(* Schneider Machine Expert - Basic project Bex CT 03 August 2023, file version 2.8.0.0 *)
(* ProjectInformations: Name=New project *)

HARDWARE
  Cpu 0: TM221CE40R
  EthernetConfiguration: NetworkName=M221, IpAllocationMode=FixedAddress, IpAddress=192.168.1.10, SubnetMask=255.255.255.0
  SerialLineConfiguration: Baud=Baud19200, Parity=ParityEven, DataBits=DataBits8, StopBits=StopBits1, PhysicalMedium=PhysicalMediumRs232, TransmissionMode=TransmissionModeModbusRtu, SlaveId=1, Addressing=MasterAddressing
  MastTask: UsePeriodScanMode=false, PeriodScan=100
  FastTask: Period=255
  CpuBehavior: StartingMode=StartAsPreviousState, AutoSaveRamOnEeprom=true, WatchdogPeriod=250

SYMBOLS  (address, symbol, comment, settings)
  %M0       SU_ALARM_AUX  "START UP ALARM AUX BIT"
  %M1       TRIP_ALARM_AUX  "SAFTY ALARM AUX BIT"
  %M2       C1_TRIP  "CONVEYOR No1 VSD TRIP"
  %M3       C2_TRIP  "CONVEYOR No2 VSD TRIP"
  %M4       SC1_TRIP  "SCALE CONVEYOR No1 VSD TRIP"
  %M5       SC1_FAULT_CONT  "SCALE CONTROL FAULT"
  %M6       C3_TRIP  "CONVEYOR No3 VSD TRIP"
  %M7       NO_PROD_STOP  "NO PRODUCT ON CONVEYOR 1 FOR PRE SET TIME"
  %M8       STOP_AUX_BIT  "STOP SEQUENCE ENERGISED"
  %M9       E_STOP_BIT  "EMERGENCY STOP AUX BIT"
  %M10      HEALTHY_BIT  "SYSTEM HEALTHY"
  %M11      C1_AUTO_START  "CONVEYOR 1 AUTO START BIT"
  %M12      C2_AUTO_START  "CONVEYOR 2 AUTO START BIT"
  %M13      SC1_AUTO_START  "SCALE CONVEYOR 1 AUTO START BIT"
  %M14      C3_AUTO_START  "CONVEYOR 3 AUTO START BIT"
  %M15      SYY_AUTO_ON  "SYSTEM AUTO RUNNING"
  %M16      C2_AUTO_STOP  "CONVEYOR 2 AUTO STOP BIT"
  %M17      SC1_AUTO_STOP  "SCALE CONVEYOR 1 AUTO STOP BIT"
  %M18      C3_AUTO_STOP  "CONVEYOR 3 AUTO STOP BIT"
  %M19      AUTO_ON_STOP  "AUTO STOP SEQUENCE ON"
  %M20      C1_ON_AUX  "C1 CONTROL BIT FULL SPEED"
  %M21      C1_ON_SLOW_AUX  "C1 CONTROL BIT SLOW SPEED"
  %M22      C2_ON_AUX  "C2 CONTROL BIT FULL SPEED"
  %M23      SC1_ON_AUX  "SC1 CONTROL BIT FULL SPEED"
  %M24      C3_ON_AUX  "C3 CONTROL BIT FULL SPEED"
  %M25      BAD_READ_AUX  "PRODUCT NOT SCANED"
  %M26      C1A_FAULT  "C1 PHOTO CELL NOT WORKING"
  %M27      C2A_FAULT  "C2 PHOTO CELL NOT WORKING"
  %M28      SC1A_FAULT  "SC1 PHOTO CELL NOT WORKING"
  %M29      C3A_FAULT  "C3 PHOTO CELL NOT WORKING"
  %M30      C1_PROD_TO_CLOSE  "PRODUCT TO CLOSED ON C1"
  %M31      C1_RESTART_PTC  "RESTART C1 AFTER PRODUCT HAS RECH CORECT DISTANCE"
  %M32      C2_PROD_TO_CLOSED  "PRODUCT TO CLOSED ON C2"
  %M33      C2_RESTART_PTC  "RESTART C2 AFTER PRODUCT HAS RECH CORECT DISTANCE"
  %M34      C1_RESTART_DELAY_C2  "RESTART C1 AFTER C2 START - TIME DELAY BIT"
  %M35      C1_RESTART_C2  "RESTART C1 AFTER C2 START - COMMAND BIT"
  %M36      SYS_RESTART_AFTER_BAD_READ  "SYSTEM RESTARTING AFTER BAD READ - AUX BIT"
  %M37      RESET_COUNTER_2  "RESET BIT FOR PRODUCT DISTANCE ON C2"
  %M38      C1A_SET_BIT  "PRODUCT COUNTER ON C1 (DISTANCE OF THE PRODUCT)"
  %M39      C2A_SET_BIT  "PRODUCT COUNTER ON C2 (DISTANCE OF THE PRODUCT)"
  %M40      APP_ON  "SIGNAL SEND FROM PC - APP ON"
  %M41      GOOD_READ_HSCAN  "SIGNAL SEND FROM THE PC - HAND SCAN GOOD READ AUX BIT"
  %M42      STOP_RUN_MSG
  %M43      HS_RESTART  "SCANING THE PRODUCT WITH HAND SCAN - GOOD READ"
  %M44      C3_BAD_READ_DELAY
  %M45      SC1A_ACTIVE_AUX1
  %M46      SCALE_EMPTY
  %M47      C1_RESTART_TIME_OUT
  %M48      C1_C2_STOP_INTERLOCK
  %M49      CF_STO_BIT
  %M50      RUN_IND
  %M51      STOP_IND
  %M52      SCALE_EMPTY_AUX
  %M53      SCALE_EMPTY_AUX1
  %M54      APP_ON_SUP_DELAY
  %M55      C2A_ACTIVE_AUX
  %M56      C2A_ACTIVE_RESET
  %M57      BAD_READ_AL
  %M58      BAD_READ_AL_AUX
  %M59      APP_SUP_DELAY_STOP
  %M60      C2_STOP_BAD_READ
  %M61      C1_STOP_BAD_READ
  %M255     BA_PASS_BIT
  %S6       SB_TB1S  "Time base of 1 s generated by an internal clock"
  %S112     SB_IOSCANETHRESET  "Set to 1 to reset the IOScanner on Ethernet"
  %SW212    SW_IOSCANETHSTATUS  "Contains the IOScanner status on Ethernet"
  %MW10     FAULT_ALARM_01  "TRIP/ALARM  SIGNALS SEND TO PC"
  %MW11     RUN_STOP_TO_PC  "SYSTEM RUNNING / STOP   SIGNALS SEND TO PC"
  %MW12     SC1A_TO_PC  "SCALE PHOTO SENSOR SC1A SIGNAL SEND TO PC"
  %MW14     PC_ON_RECEIVED
  %MW20     RECEIVED_FROM_PC_ON  "SIGNAL SEND FROM PC - PC ON"
  %MW25     RECEIVED_FROM_PC_HSGR  "SIGNAL RECEIVED FROM PC - HAND SCAN GOOD READ"
  %TM0        [Preset=14, Base=OneSecond]
  %TM1        [Preset=10]
  %TM2        [Preset=25, Base=OneSecond]
  %TM3        [Preset=100, Base=OneSecond]
  %TM4        [Preset=1, Base=OneSecond]
  %TM5        [Preset=1, Base=OneSecond]
  %TM6        [Preset=5, Base=TenMilliSeconds]
  %TM7        [Preset=2, Base=TenMilliSeconds]
  %TM8        [Preset=180, Base=OneSecond]
  %TM9        [Preset=180, Base=OneSecond]
  %TM10       [Preset=180, Base=OneSecond]
  %TM11       [Preset=120, Base=OneSecond]
  %TM12       [Preset=1, Base=OneSecond]
  %TM13       [Preset=30, Base=TenMilliSeconds]
  %TM14       [Preset=3, Base=OneSecond]
  %TM15       [Type=TOF, Preset=120, Base=OneSecond]
  %TM16       [Preset=1, Base=TenMilliSeconds]
  %TM17       [Preset=3, Base=OneSecond]
  %TM18       [Preset=3, Base=OneSecond]
  %TM19       [Preset=5, Base=TenMilliSeconds]
  %TM20       [Preset=5, Base=TenMilliSeconds]
  %C0         [Preset=2]
  %C1         [Preset=2]
  %I0.0     E_STOP_PB  "EMERGENCY STOP PUSH BUTTON"
  %I0.1     SYS_START_PB  "Alarm Acknowledge Push Button"
  %I0.2     SYS_STOP_PB  "Alarm Reset Push Button"
  %I0.3     ALARM_ACKG  "System Start Push Button"
  %I0.4     ALARM_RESET  "System Stop Push Button"
  %I0.5     C1_RUNNING  "Conveyor No.1 Running  VSD"
  %I0.6     C2_RUNNING  "Conveyor No.2 Running  VSD"
  %I0.7     SC1_RUNNING  "Scale Conveyor No.1 Running  VSD"
  %I0.8     C3_RUNNING  "Conveyor No.3 Running  VSD"
  %I0.9     C1A_ACTIVE  "Conveyor No.1 Photo Sensor"
  %I0.10    C2A_ACTIVE  "Conveyor No.2 Photo Sensor"
  %I0.11    SC1A_ACTIVE  "Scale Conveyor No.1 Photo Sensor"
  %I0.12    SC1B_ACTIVE  "Scale Conveyor No.1  Control Fault"
  %I0.13    C3A_ACTIVE  "Conveyor No.3 Photo Sensor"
  %I0.14    GOOD_READ_ACTIVE  "Camera Product Good Read"
  %I0.15    BAD_READ_ACTIVE  "Camera Product Bad Read"
  %I0.16    LASER_READ  "LASER SIGNAL IN"
  %I0.17    CAMERA_SENS  "CAMERA SENSOR ON SCALE CONVEYOR"
  %Q0.0     C1_ON  "Conveyor No.1 - ON/OFF Fast"
  %Q0.1     C1_ON_SLOW  "Conveyor No.1 - SLOW SPEED"
  %Q0.2     C2_ON  "Conveyor No.2 - ON/OFF Fast"
  %Q0.3     C2_ON_SLOW  "Conveyor No.2 - SLOW SPEED"
  %Q0.4     SC1_ON  "Scale belt No.1 - ON/OFF Fast"
  %Q0.5     SC1_ON_SLOW  "Scale belt No.1 - SLOW SPEED"
  %Q0.6     C3_ON  "ConveConveyor No.3 - ON/OFF Fast"
  %Q0.7     C3_ON_SLOW  "Conveyor No.3 - SLOW SPEED"
  %Q0.8     SYS_RUNNING_IND  "System Running Green Indication"
  %Q0.9     SYS_TRIP_IND  "System Trip Red Indication"
  %Q0.10    ALARM_BUZZER  "Alarm Buzzer"
  %Q0.11    GOOD_READ_IND  "Product Good read Tower Green indication"
  %Q0.12    BAD_READ_IND  "Product Bad read Tower Green indication"
  %Q0.13    SC1_CONT_ON  "Start Scale - Signal to Scale Control  Panel"
  %Q0.14    CAM_TRIGGER  "Camera On/Off with laser or Sensor on the scale belt"
  %Q0.15    COLLING_FAN
  %IWN300.0.0 PC_IN_01  "APPLICATION RUNNING / STOP SIGNAL SEND FROM THE PC"  [Channel=Device 1_Channel0]
  %IWN300.0.1 PC_IN_02  "HAND SCANER ON/OFF SIGNAL SEND FROM PC"  [Channel=Device 1_Channel0]
  %QWN300.1.0 PC_OUT_01  "SENDING TO PC - ALARMS"  [Channel=Device 1_Channel1]
  %QWN300.1.1 PC_OUT_02  "SENDING TO PC STATUS (RUN, STOP, E/STOP)"  [Channel=Device 1_Channel1]
  %QWN300.1.2 PC_OUT_03  "SENDING TO PC - SCALE PHOTO SENSOR STATUS"  [Channel=Device 1_Channel1]
  %QWN300.1.3 PC_OUT_04  [Channel=Device 1_Channel1]

POU GENERAL ALARM
  (* SectionNumber=1 *)

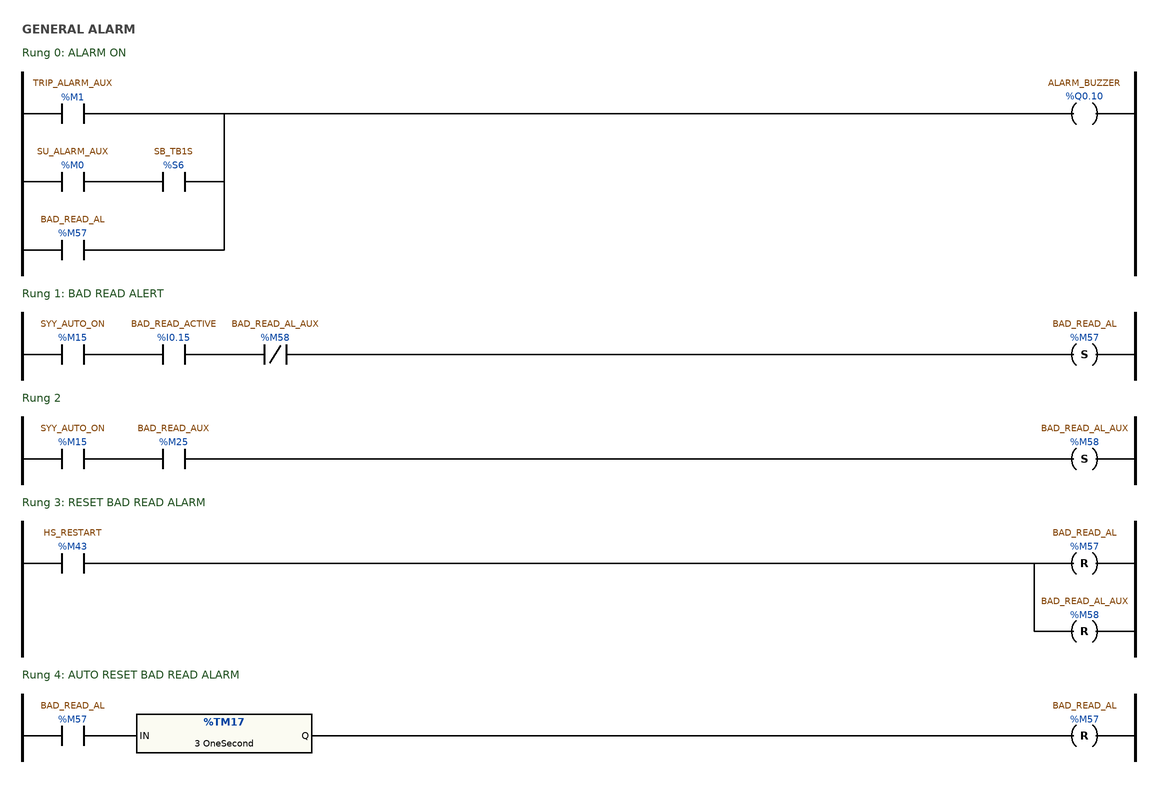

// Rung 0: ALARM ON
  LD %M1                  (* TRIP_ALARM_AUX *)
  OR( %M0                 (* SU_ALARM_AUX *)
  AND %S6                 (* SB_TB1S *)
  )
  OR %M57                 (* BAD_READ_AL *)
  ST %Q0.10               (* ALARM_BUZZER *)
  // as ST:
  //   ALARM_BUZZER := TRIP_ALARM_AUX OR SU_ALARM_AUX AND SB_TB1S OR BAD_READ_AL;

// Rung 1: BAD READ ALERT
  LD %M15                 (* SYY_AUTO_ON *)
  AND %I0.15              (* BAD_READ_ACTIVE *)
  ANDN %M58               (* BAD_READ_AL_AUX *)
  S %M57                  (* BAD_READ_AL *)
  // as ST:
  //   IF SYY_AUTO_ON AND BAD_READ_ACTIVE AND NOT BAD_READ_AL_AUX THEN BAD_READ_AL := TRUE; END_IF;

// Rung 2
  LD %M15                 (* SYY_AUTO_ON *)
  AND %M25                (* BAD_READ_AUX *)
  S %M58                  (* BAD_READ_AL_AUX *)
  // as ST:
  //   IF SYY_AUTO_ON AND BAD_READ_AUX THEN BAD_READ_AL_AUX := TRUE; END_IF;

// Rung 3: RESET BAD READ ALARM
  LD %M43                 (* HS_RESTART *)
  R %M57                  (* BAD_READ_AL *)
  R %M58                  (* BAD_READ_AL_AUX *)
  // as ST:
  //   IF HS_RESTART THEN BAD_READ_AL := FALSE; END_IF;
  //   IF HS_RESTART THEN BAD_READ_AL_AUX := FALSE; END_IF;

// Rung 4: AUTO RESET BAD READ ALARM
  BLK %TM17
  LD %M57                 (* BAD_READ_AL *)
  IN
  OUT_BLK
  LD Q
  R %M57                  (* BAD_READ_AL *)
  END_BLK
  // as ST:
  //   %TM17(IN := BAD_READ_AL);
  //   IF %TM17.Q THEN BAD_READ_AL := FALSE; END_IF;

POU START UP ALARM
  (* SectionNumber=2 *)

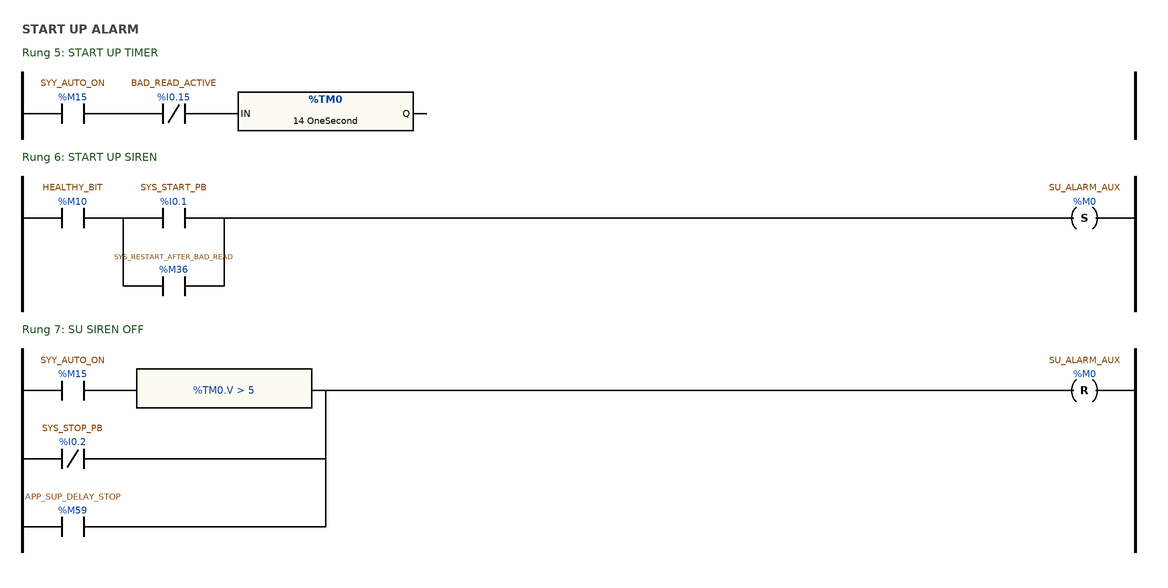

// Rung 5: START UP TIMER
  BLK %TM0
  LD %M15                 (* SYY_AUTO_ON *)
  ANDN %I0.15             (* BAD_READ_ACTIVE *)
  IN
  END_BLK
  // as ST:
  //   %TM0(IN := SYY_AUTO_ON AND NOT BAD_READ_ACTIVE);

// Rung 6: START UP SIREN
  LD %M10                 (* HEALTHY_BIT *)
  AND( %I0.1              (* SYS_START_PB *)
  OR %M36                 (* SYS_RESTART_AFTER_BAD_READ *)
  )
  S %M0                   (* SU_ALARM_AUX *)
  // as ST:
  //   IF HEALTHY_BIT AND (SYS_START_PB OR SYS_RESTART_AFTER_BAD_READ) THEN SU_ALARM_AUX := TRUE; END_IF;

// Rung 7: SU SIREN OFF
  LD %M15                 (* SYY_AUTO_ON *)
  AND [ %TM0.V > 5 ]
  ORN %I0.2               (* SYS_STOP_PB *)
  OR %M59                 (* APP_SUP_DELAY_STOP *)
  R %M0                   (* SU_ALARM_AUX *)
  // as ST:
  //   IF SYY_AUTO_ON AND %TM0.V > 5 OR NOT SYS_STOP_PB OR APP_SUP_DELAY_STOP THEN SU_ALARM_AUX := FALSE; END_IF;

POU SAFETY ALARM
  (* SectionNumber=3 *)

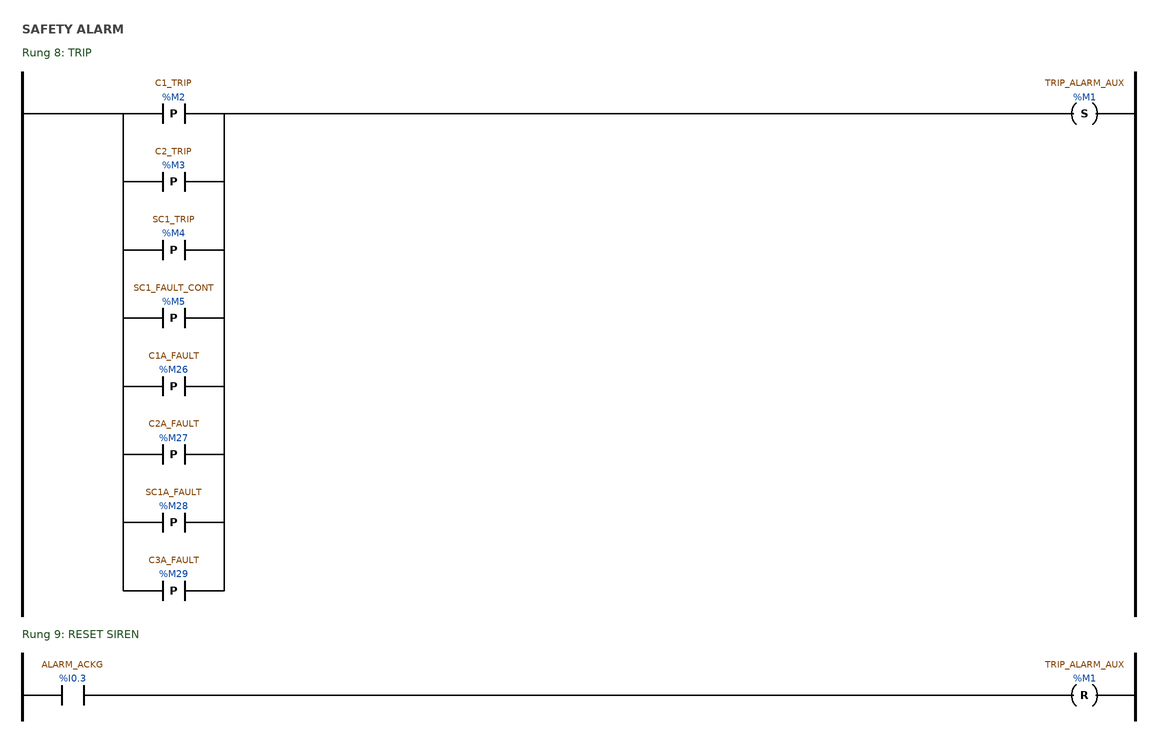

// Rung 8: TRIP
  LD 1
  AND(R %M2               (* C1_TRIP *)
  ORR %M3                 (* C2_TRIP *)
  ORR %M4                 (* SC1_TRIP *)
  ORR %M5                 (* SC1_FAULT_CONT *)
  ORR %M26                (* C1A_FAULT *)
  ORR %M27                (* C2A_FAULT *)
  ORR %M28                (* SC1A_FAULT *)
  ORR %M29                (* C3A_FAULT *)
  )
  S %M1                   (* TRIP_ALARM_AUX *)
  // as ST:
  //   IF RISING(C1_TRIP) OR RISING(C2_TRIP) OR RISING(SC1_TRIP) OR RISING(SC1_FAULT_CONT) OR RISING(C1A_FAULT) OR RISING(C2A_FAULT) OR RISING(SC1A_FAULT) OR RISING(C3A_FAULT) THEN TRIP_ALARM_AUX := TRUE; END_IF;

// Rung 9: RESET SIREN
  LD %I0.3                (* ALARM_ACKG *)
  R %M1                   (* TRIP_ALARM_AUX *)
  // as ST:
  //   IF ALARM_ACKG THEN TRIP_ALARM_AUX := FALSE; END_IF;

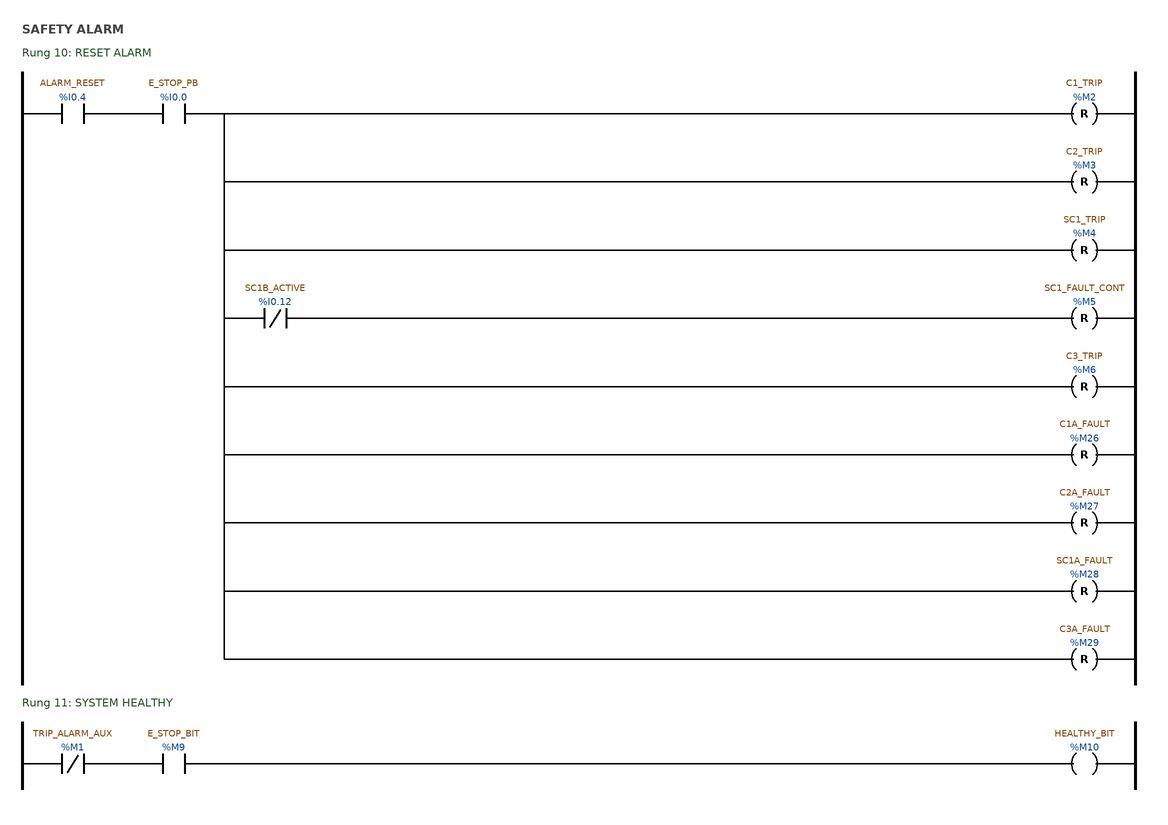

// Rung 10: RESET ALARM
  LD %I0.4                (* ALARM_RESET *)
  AND %I0.0               (* E_STOP_PB *)
  MPS
  R %M2                   (* C1_TRIP *)
  MRD
  R %M3                   (* C2_TRIP *)
  MRD
  R %M4                   (* SC1_TRIP *)
  MRD
  ANDN %I0.12             (* SC1B_ACTIVE *)
  R %M5                   (* SC1_FAULT_CONT *)
  MRD
  R %M6                   (* C3_TRIP *)
  MRD
  R %M26                  (* C1A_FAULT *)
  MRD
  R %M27                  (* C2A_FAULT *)
  MRD
  R %M28                  (* SC1A_FAULT *)
  MPP
  R %M29                  (* C3A_FAULT *)
  // as ST:
  //   IF ALARM_RESET AND E_STOP_PB THEN C1_TRIP := FALSE; END_IF;
  //   IF ALARM_RESET AND E_STOP_PB THEN C2_TRIP := FALSE; END_IF;
  //   IF ALARM_RESET AND E_STOP_PB THEN SC1_TRIP := FALSE; END_IF;
  //   IF ALARM_RESET AND E_STOP_PB AND NOT SC1B_ACTIVE THEN SC1_FAULT_CONT := FALSE; END_IF;
  //   IF ALARM_RESET AND E_STOP_PB THEN C3_TRIP := FALSE; END_IF;
  //   IF ALARM_RESET AND E_STOP_PB THEN C1A_FAULT := FALSE; END_IF;
  //   IF ALARM_RESET AND E_STOP_PB THEN C2A_FAULT := FALSE; END_IF;
  //   IF ALARM_RESET AND E_STOP_PB THEN SC1A_FAULT := FALSE; END_IF;
  //   IF ALARM_RESET AND E_STOP_PB THEN C3A_FAULT := FALSE; END_IF;

// Rung 11: SYSTEM HEALTHY
  LDN %M1                 (* TRIP_ALARM_AUX *)
  AND %M9                 (* E_STOP_BIT *)
  ST %M10                 (* HEALTHY_BIT *)
  // as ST:
  //   HEALTHY_BIT := NOT TRIP_ALARM_AUX AND E_STOP_BIT;

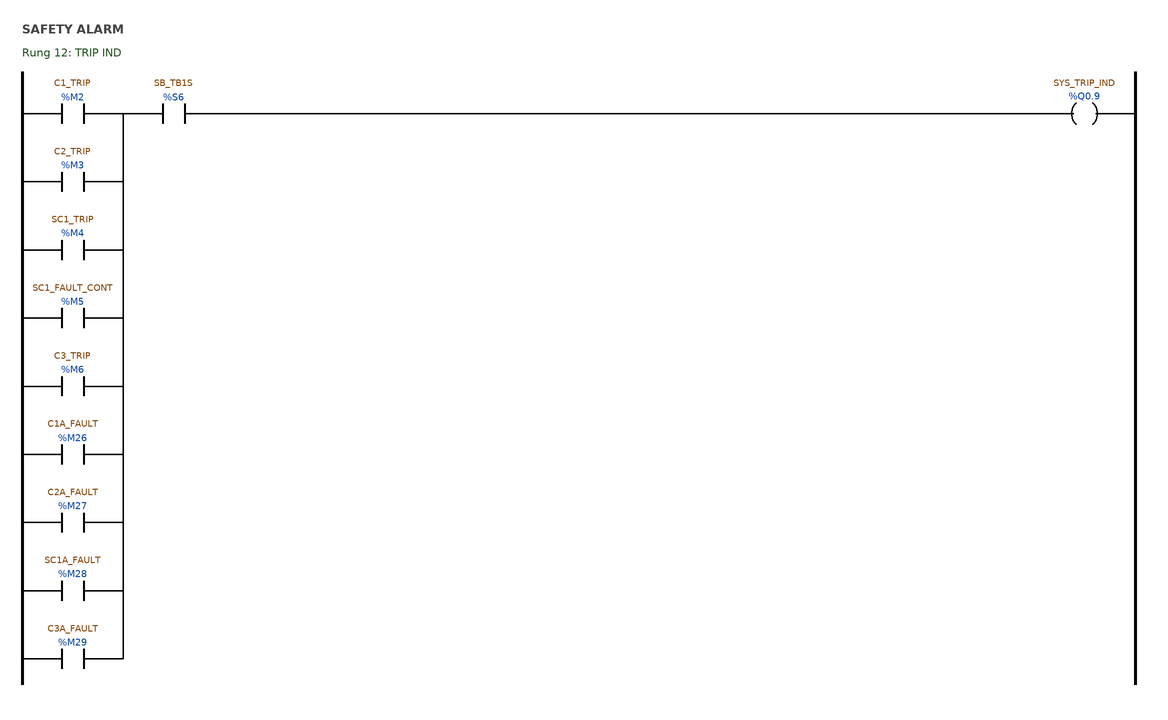

// Rung 12: TRIP IND
  LD %M2                  (* C1_TRIP *)
  OR %M3                  (* C2_TRIP *)
  OR %M4                  (* SC1_TRIP *)
  OR %M5                  (* SC1_FAULT_CONT *)
  OR %M6                  (* C3_TRIP *)
  OR %M26                 (* C1A_FAULT *)
  OR %M27                 (* C2A_FAULT *)
  OR %M28                 (* SC1A_FAULT *)
  OR %M29                 (* C3A_FAULT *)
  AND %S6                 (* SB_TB1S *)
  ST %Q0.9                (* SYS_TRIP_IND *)
  // as ST:
  //   SYS_TRIP_IND := (C1_TRIP OR C2_TRIP OR SC1_TRIP OR SC1_FAULT_CONT OR C3_TRIP OR C1A_FAULT OR C2A_FAULT OR SC1A_FAULT OR C3A_FAULT) AND SB_TB1S;

POU SENSORS FAULT
  (* SectionNumber=4 *)

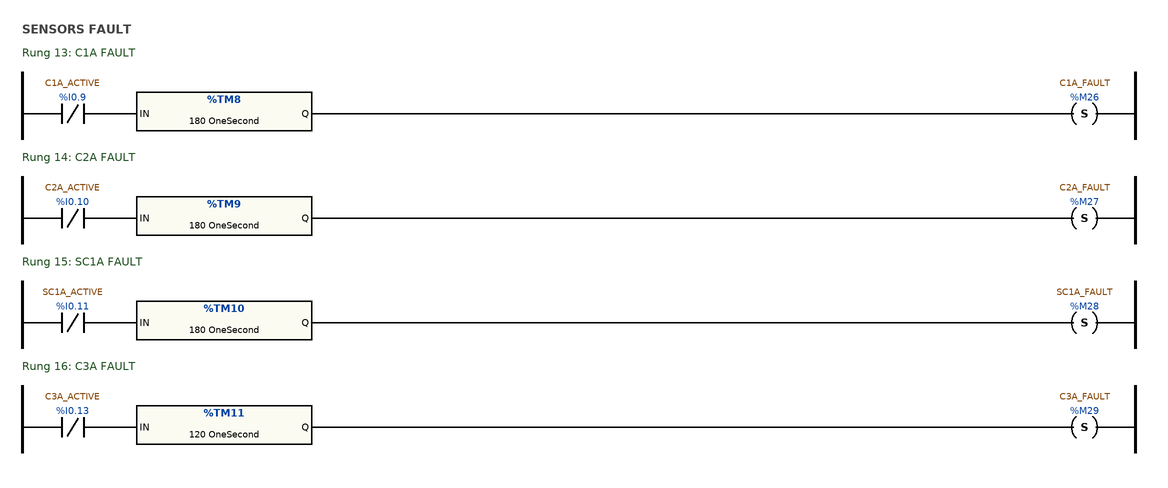

// Rung 13: C1A FAULT
  BLK %TM8
  LDN %I0.9               (* C1A_ACTIVE *)
  IN
  OUT_BLK
  LD Q
  S %M26                  (* C1A_FAULT *)
  END_BLK
  // as ST:
  //   %TM8(IN := NOT C1A_ACTIVE);
  //   IF %TM8.Q THEN C1A_FAULT := TRUE; END_IF;

// Rung 14: C2A FAULT
  BLK %TM9
  LDN %I0.10              (* C2A_ACTIVE *)
  IN
  OUT_BLK
  LD Q
  S %M27                  (* C2A_FAULT *)
  END_BLK
  // as ST:
  //   %TM9(IN := NOT C2A_ACTIVE);
  //   IF %TM9.Q THEN C2A_FAULT := TRUE; END_IF;

// Rung 15: SC1A FAULT
  BLK %TM10
  LDN %I0.11              (* SC1A_ACTIVE *)
  IN
  OUT_BLK
  LD Q
  S %M28                  (* SC1A_FAULT *)
  END_BLK
  // as ST:
  //   %TM10(IN := NOT SC1A_ACTIVE);
  //   IF %TM10.Q THEN SC1A_FAULT := TRUE; END_IF;

// Rung 16: C3A FAULT
  BLK %TM11
  LDN %I0.13              (* C3A_ACTIVE *)
  IN
  OUT_BLK
  LD Q
  S %M29                  (* C3A_FAULT *)
  END_BLK
  // as ST:
  //   %TM11(IN := NOT C3A_ACTIVE);
  //   IF %TM11.Q THEN C3A_FAULT := TRUE; END_IF;

POU CONTROL
  (* SectionNumber=5 *)

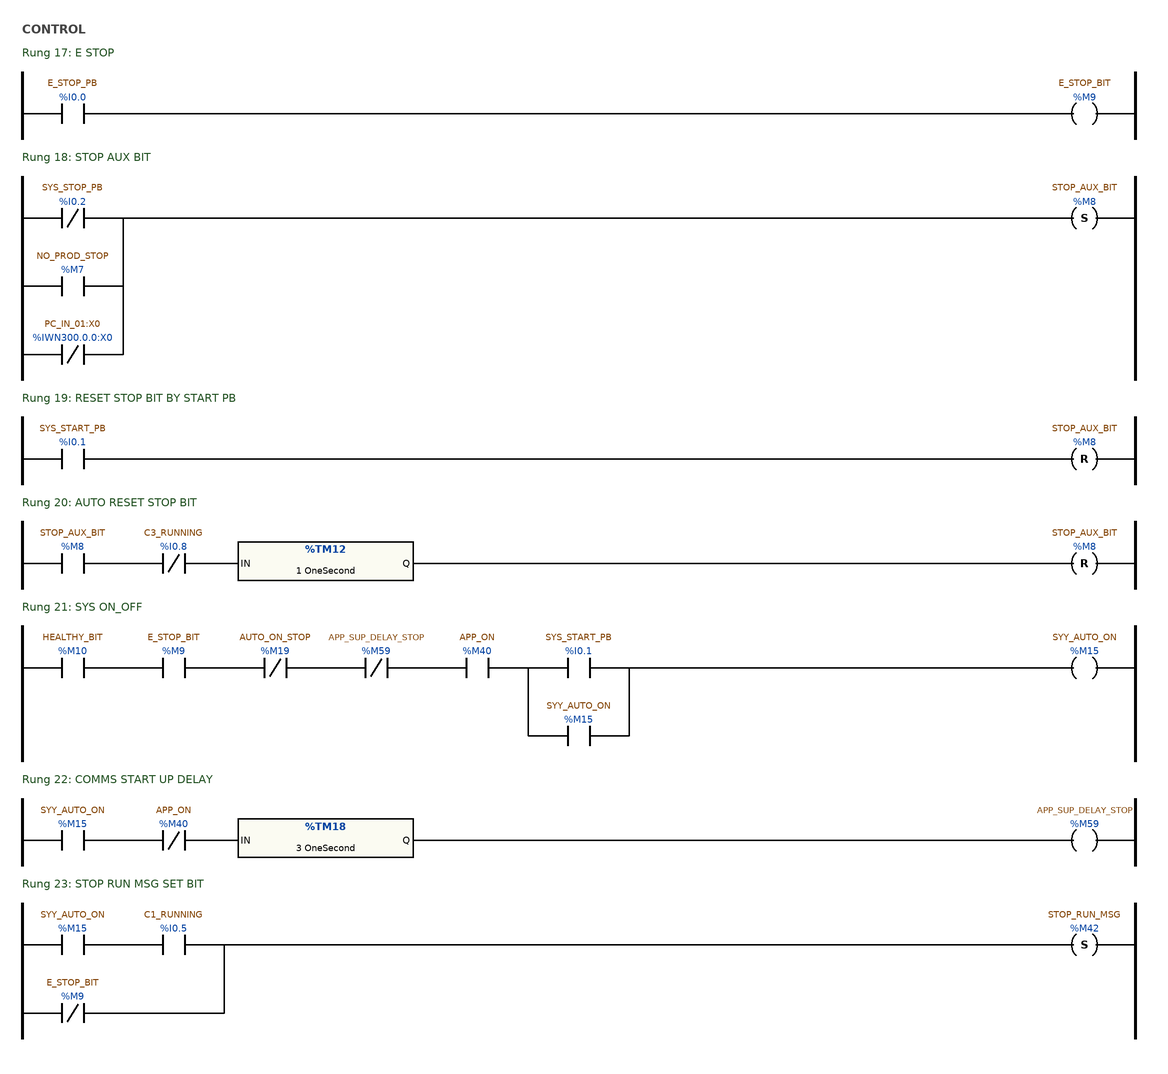

// Rung 17: E STOP
  LD %I0.0                (* E_STOP_PB *)
  ST %M9                  (* E_STOP_BIT *)
  // as ST:
  //   E_STOP_BIT := E_STOP_PB;

// Rung 18: STOP AUX BIT
  LDN %I0.2               (* SYS_STOP_PB *)
  OR %M7                  (* NO_PROD_STOP *)
  ORN %IWN300.0.0:X0      (* PC_IN_01 *)
  S %M8                   (* STOP_AUX_BIT *)
  // as ST:
  //   IF NOT SYS_STOP_PB OR NO_PROD_STOP OR NOT PC_IN_01:X0 THEN STOP_AUX_BIT := TRUE; END_IF;

// Rung 19: RESET STOP BIT BY START PB
  LD %I0.1                (* SYS_START_PB *)
  R %M8                   (* STOP_AUX_BIT *)
  // as ST:
  //   IF SYS_START_PB THEN STOP_AUX_BIT := FALSE; END_IF;

// Rung 20: AUTO RESET STOP BIT
  BLK %TM12
  LD %M8                  (* STOP_AUX_BIT *)
  ANDN %I0.8              (* C3_RUNNING *)
  IN
  OUT_BLK
  LD Q
  R %M8                   (* STOP_AUX_BIT *)
  END_BLK
  // as ST:
  //   %TM12(IN := STOP_AUX_BIT AND NOT C3_RUNNING);
  //   IF %TM12.Q THEN STOP_AUX_BIT := FALSE; END_IF;

// Rung 21: SYS ON_OFF
  LD %M10                 (* HEALTHY_BIT *)
  AND %M9                 (* E_STOP_BIT *)
  ANDN %M19               (* AUTO_ON_STOP *)
  ANDN %M59               (* APP_SUP_DELAY_STOP *)
  AND %M40                (* APP_ON *)
  AND( %I0.1              (* SYS_START_PB *)
  OR %M15                 (* SYY_AUTO_ON *)
  )
  ST %M15                 (* SYY_AUTO_ON *)
  // as ST:
  //   SYY_AUTO_ON := HEALTHY_BIT AND E_STOP_BIT AND NOT AUTO_ON_STOP AND NOT APP_SUP_DELAY_STOP AND APP_ON AND (SYS_START_PB OR SYY_AUTO_ON);

// Rung 22: COMMS START UP DELAY
  BLK %TM18
  LD %M15                 (* SYY_AUTO_ON *)
  ANDN %M40               (* APP_ON *)
  IN
  OUT_BLK
  LD Q
  ST %M59                 (* APP_SUP_DELAY_STOP *)
  END_BLK
  // as ST:
  //   %TM18(IN := SYY_AUTO_ON AND NOT APP_ON);
  //   APP_SUP_DELAY_STOP := %TM18.Q;

// Rung 23: STOP RUN MSG SET BIT
  LD %M15                 (* SYY_AUTO_ON *)
  AND %I0.5               (* C1_RUNNING *)
  ORN %M9                 (* E_STOP_BIT *)
  S %M42                  (* STOP_RUN_MSG *)
  // as ST:
  //   IF SYY_AUTO_ON AND C1_RUNNING OR NOT E_STOP_BIT THEN STOP_RUN_MSG := TRUE; END_IF;

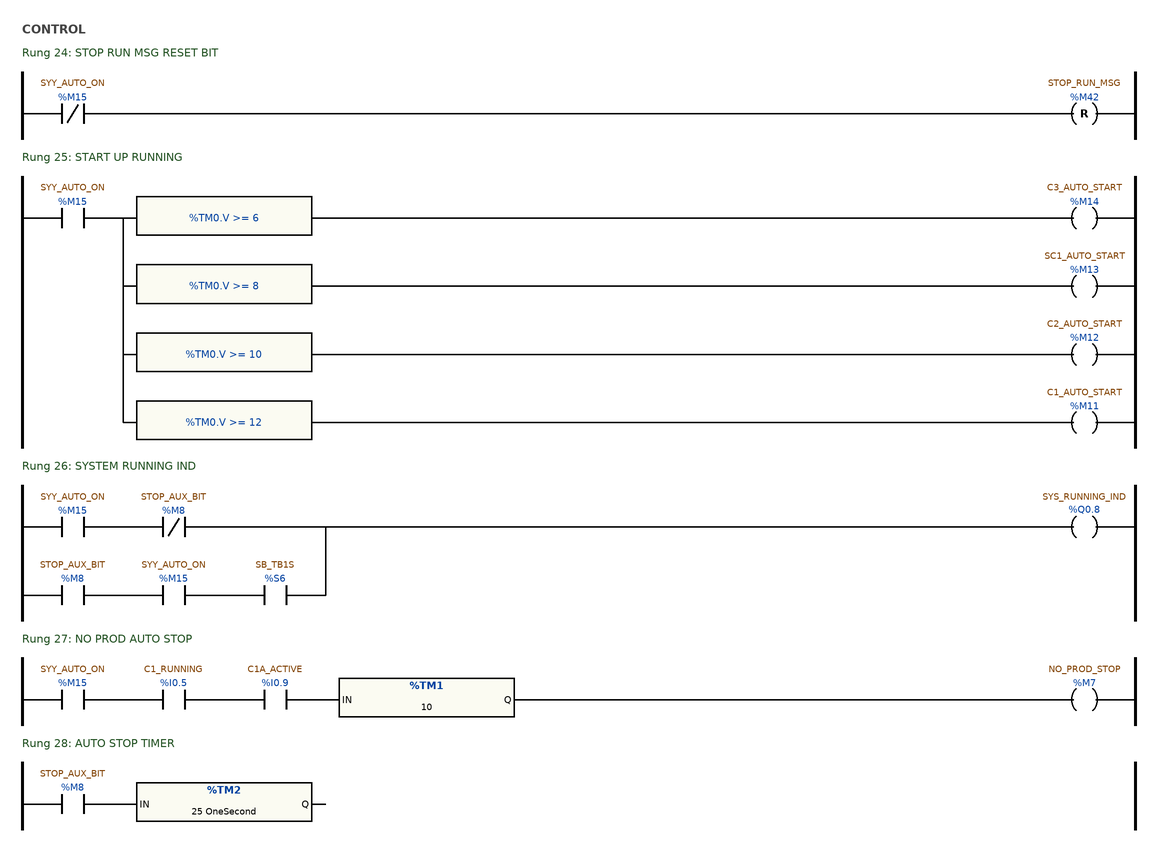

// Rung 24: STOP RUN MSG RESET BIT
  LDN %M15                (* SYY_AUTO_ON *)
  R %M42                  (* STOP_RUN_MSG *)
  // as ST:
  //   IF NOT SYY_AUTO_ON THEN STOP_RUN_MSG := FALSE; END_IF;

// Rung 25: START UP RUNNING
  LD %M15                 (* SYY_AUTO_ON *)
  MPS
  AND [ %TM0.V >= 6 ]
  ST %M14                 (* C3_AUTO_START *)
  MRD
  AND [ %TM0.V >= 8 ]
  ST %M13                 (* SC1_AUTO_START *)
  MRD
  AND [ %TM0.V >= 10 ]
  ST %M12                 (* C2_AUTO_START *)
  MPP
  AND [ %TM0.V >= 12 ]
  ST %M11                 (* C1_AUTO_START *)
  // as ST:
  //   C3_AUTO_START := SYY_AUTO_ON AND %TM0.V >= 6;
  //   SC1_AUTO_START := SYY_AUTO_ON AND %TM0.V >= 8;
  //   C2_AUTO_START := SYY_AUTO_ON AND %TM0.V >= 10;
  //   C1_AUTO_START := SYY_AUTO_ON AND %TM0.V >= 12;

// Rung 26: SYSTEM RUNNING IND
  LD %M15                 (* SYY_AUTO_ON *)
  ANDN %M8                (* STOP_AUX_BIT *)
  OR( %M8                 (* STOP_AUX_BIT *)
  AND %M15                (* SYY_AUTO_ON *)
  AND %S6                 (* SB_TB1S *)
  )
  ST %Q0.8                (* SYS_RUNNING_IND *)
  // as ST:
  //   SYS_RUNNING_IND := SYY_AUTO_ON AND NOT STOP_AUX_BIT OR STOP_AUX_BIT AND SYY_AUTO_ON AND SB_TB1S;

// Rung 27: NO PROD AUTO STOP
  BLK %TM1
  LD %M15                 (* SYY_AUTO_ON *)
  AND %I0.5               (* C1_RUNNING *)
  AND %I0.9               (* C1A_ACTIVE *)
  IN
  OUT_BLK
  LD Q
  ST %M7                  (* NO_PROD_STOP *)
  END_BLK
  // as ST:
  //   %TM1(IN := SYY_AUTO_ON AND C1_RUNNING AND C1A_ACTIVE);
  //   NO_PROD_STOP := %TM1.Q;

// Rung 28: AUTO STOP TIMER
  BLK %TM2
  LD %M8                  (* STOP_AUX_BIT *)
  IN
  END_BLK
  // as ST:
  //   %TM2(IN := STOP_AUX_BIT);

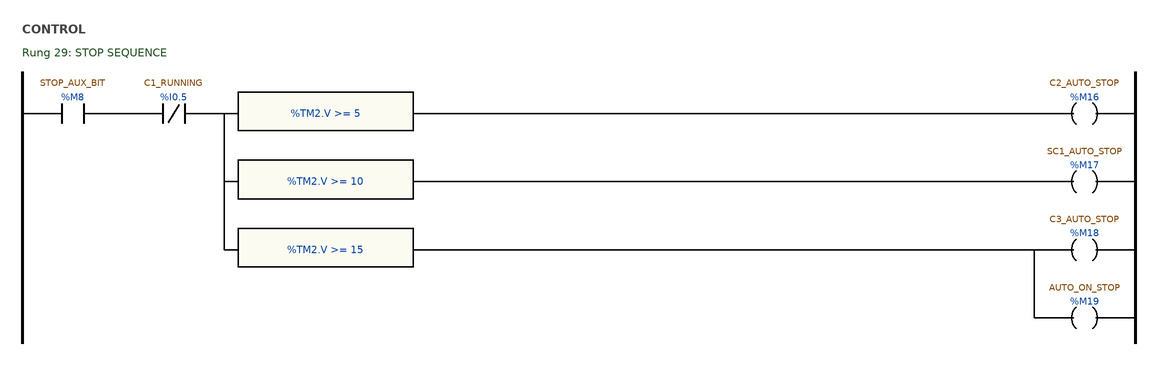

// Rung 29: STOP SEQUENCE
  LD %M8                  (* STOP_AUX_BIT *)
  ANDN %I0.5              (* C1_RUNNING *)
  MPS
  AND [ %TM2.V >= 5 ]
  ST %M16                 (* C2_AUTO_STOP *)
  MRD
  AND [ %TM2.V >= 10 ]
  ST %M17                 (* SC1_AUTO_STOP *)
  MPP
  AND [ %TM2.V >= 15 ]
  ST %M18                 (* C3_AUTO_STOP *)
  ST %M19                 (* AUTO_ON_STOP *)
  // as ST:
  //   C2_AUTO_STOP := STOP_AUX_BIT AND NOT C1_RUNNING AND %TM2.V >= 5;
  //   SC1_AUTO_STOP := STOP_AUX_BIT AND NOT C1_RUNNING AND %TM2.V >= 10;
  //   C3_AUTO_STOP := STOP_AUX_BIT AND NOT C1_RUNNING AND %TM2.V >= 15;
  //   AUTO_ON_STOP := STOP_AUX_BIT AND NOT C1_RUNNING AND %TM2.V >= 15;

POU CONVEYOR No1
  (* SectionNumber=6 *)

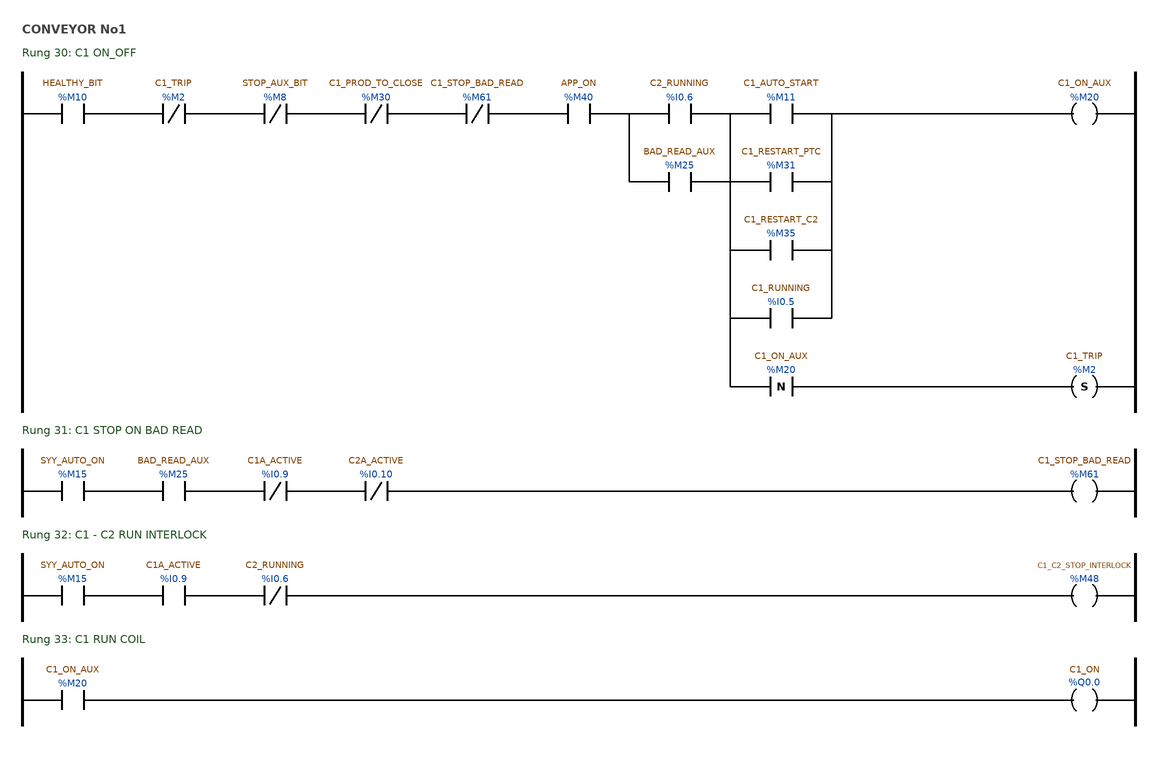

// Rung 30: C1 ON_OFF
  LD %M10                 (* HEALTHY_BIT *)
  ANDN %M2                (* C1_TRIP *)
  ANDN %M8                (* STOP_AUX_BIT *)
  ANDN %M30               (* C1_PROD_TO_CLOSE *)
  ANDN %M61               (* C1_STOP_BAD_READ *)
  AND %M40                (* APP_ON *)
  AND( %I0.6              (* C2_RUNNING *)
  OR %M25                 (* BAD_READ_AUX *)
  )
  MPS
  AND( %M11               (* C1_AUTO_START *)
  OR %M31                 (* C1_RESTART_PTC *)
  OR %M35                 (* C1_RESTART_C2 *)
  OR %I0.5                (* C1_RUNNING *)
  )
  ST %M20                 (* C1_ON_AUX *)
  MPP
  ANDF %M20               (* C1_ON_AUX *)
  S %M2                   (* C1_TRIP *)
  // as ST:
  //   C1_ON_AUX := HEALTHY_BIT AND NOT C1_TRIP AND NOT STOP_AUX_BIT AND NOT C1_PROD_TO_CLOSE AND NOT C1_STOP_BAD_READ AND APP_ON AND (C2_RUNNING OR BAD_READ_AUX) AND (C1_AUTO_START OR C1_RESTART_PTC OR C1_RESTART_C2 OR C1_RUNNING);
  //   IF HEALTHY_BIT AND NOT C1_TRIP AND NOT STOP_AUX_BIT AND NOT C1_PROD_TO_CLOSE AND NOT C1_STOP_BAD_READ AND APP_ON AND (C2_RUNNING OR BAD_READ_AUX) AND FALLING(C1_ON_AUX) THEN C1_TRIP := TRUE; END_IF;

// Rung 31: C1 STOP ON BAD READ
  LD %M15                 (* SYY_AUTO_ON *)
  AND %M25                (* BAD_READ_AUX *)
  ANDN %I0.9              (* C1A_ACTIVE *)
  ANDN %I0.10             (* C2A_ACTIVE *)
  ST %M61                 (* C1_STOP_BAD_READ *)
  // as ST:
  //   C1_STOP_BAD_READ := SYY_AUTO_ON AND BAD_READ_AUX AND NOT C1A_ACTIVE AND NOT C2A_ACTIVE;

// Rung 32: C1 - C2 RUN INTERLOCK
  LD %M15                 (* SYY_AUTO_ON *)
  AND %I0.9               (* C1A_ACTIVE *)
  ANDN %I0.6              (* C2_RUNNING *)
  ST %M48                 (* C1_C2_STOP_INTERLOCK *)
  // as ST:
  //   C1_C2_STOP_INTERLOCK := SYY_AUTO_ON AND C1A_ACTIVE AND NOT C2_RUNNING;

// Rung 33: C1 RUN COIL
  LD %M20                 (* C1_ON_AUX *)
  ST %Q0.0                (* C1_ON *)
  // as ST:
  //   C1_ON := C1_ON_AUX;

POU CONVEYOR No2
  (* SectionNumber=7 *)

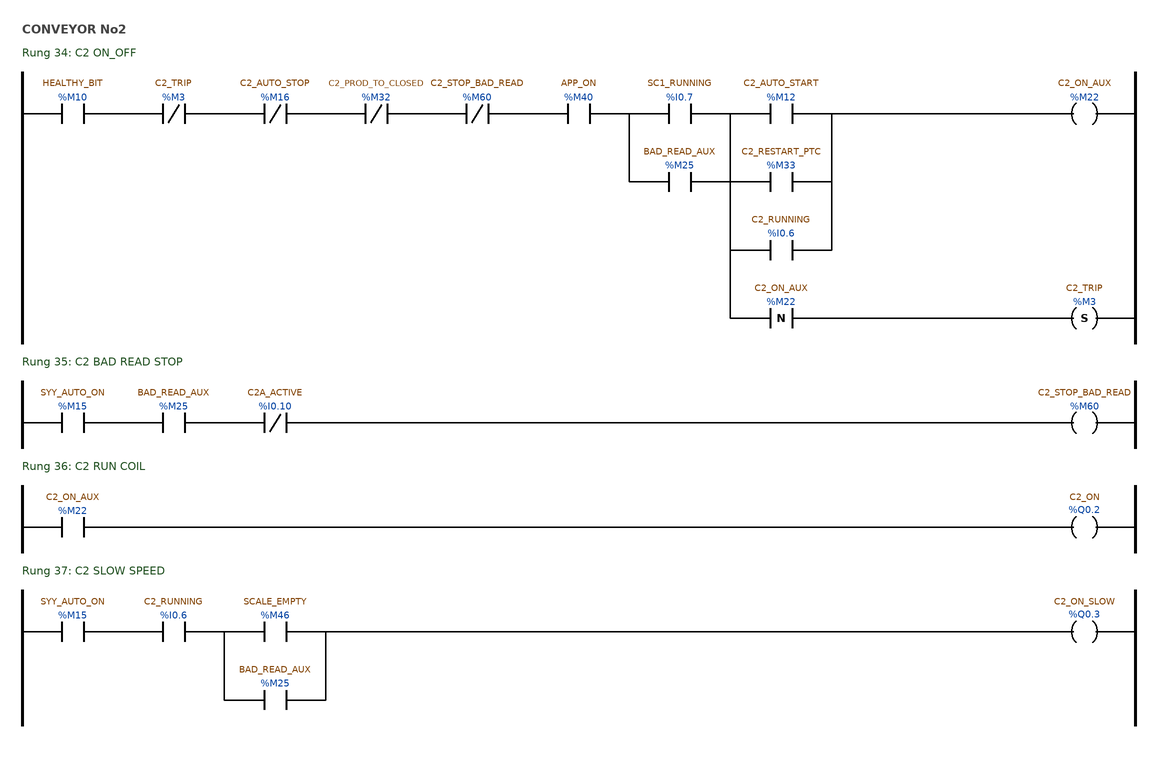

// Rung 34: C2 ON_OFF
  LD %M10                 (* HEALTHY_BIT *)
  ANDN %M3                (* C2_TRIP *)
  ANDN %M16               (* C2_AUTO_STOP *)
  ANDN %M32               (* C2_PROD_TO_CLOSED *)
  ANDN %M60               (* C2_STOP_BAD_READ *)
  AND %M40                (* APP_ON *)
  AND( %I0.7              (* SC1_RUNNING *)
  OR %M25                 (* BAD_READ_AUX *)
  )
  MPS
  AND( %M12               (* C2_AUTO_START *)
  OR %M33                 (* C2_RESTART_PTC *)
  OR %I0.6                (* C2_RUNNING *)
  )
  ST %M22                 (* C2_ON_AUX *)
  MPP
  ANDF %M22               (* C2_ON_AUX *)
  S %M3                   (* C2_TRIP *)
  // as ST:
  //   C2_ON_AUX := HEALTHY_BIT AND NOT C2_TRIP AND NOT C2_AUTO_STOP AND NOT C2_PROD_TO_CLOSED AND NOT C2_STOP_BAD_READ AND APP_ON AND (SC1_RUNNING OR BAD_READ_AUX) AND (C2_AUTO_START OR C2_RESTART_PTC OR C2_RUNNING);
  //   IF HEALTHY_BIT AND NOT C2_TRIP AND NOT C2_AUTO_STOP AND NOT C2_PROD_TO_CLOSED AND NOT C2_STOP_BAD_READ AND APP_ON AND (SC1_RUNNING OR BAD_READ_AUX) AND FALLING(C2_ON_AUX) THEN C2_TRIP := TRUE; END_IF;

// Rung 35: C2 BAD READ STOP
  LD %M15                 (* SYY_AUTO_ON *)
  AND %M25                (* BAD_READ_AUX *)
  ANDN %I0.10             (* C2A_ACTIVE *)
  ST %M60                 (* C2_STOP_BAD_READ *)
  // as ST:
  //   C2_STOP_BAD_READ := SYY_AUTO_ON AND BAD_READ_AUX AND NOT C2A_ACTIVE;

// Rung 36: C2 RUN COIL
  LD %M22                 (* C2_ON_AUX *)
  ST %Q0.2                (* C2_ON *)
  // as ST:
  //   C2_ON := C2_ON_AUX;

// Rung 37: C2 SLOW SPEED
  LD %M15                 (* SYY_AUTO_ON *)
  AND %I0.6               (* C2_RUNNING *)
  AND( %M46               (* SCALE_EMPTY *)
  OR %M25                 (* BAD_READ_AUX *)
  )
  ST %Q0.3                (* C2_ON_SLOW *)
  // as ST:
  //   C2_ON_SLOW := SYY_AUTO_ON AND C2_RUNNING AND (SCALE_EMPTY OR BAD_READ_AUX);

POU SCALE No1
  (* SectionNumber=8 *)

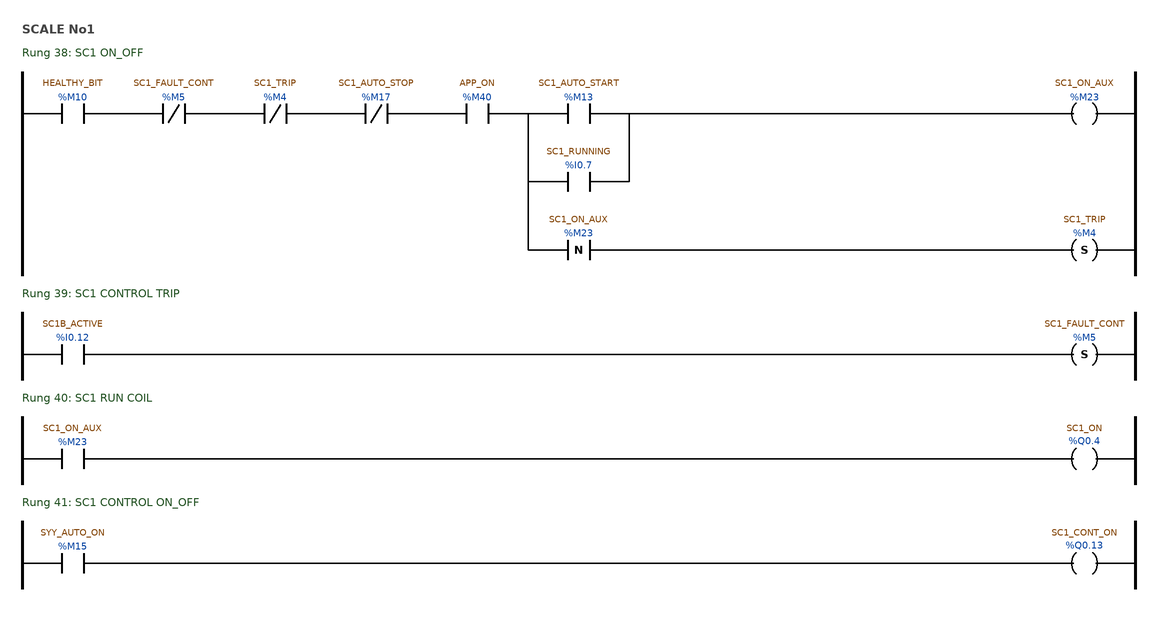

// Rung 38: SC1 ON_OFF
  LD %M10                 (* HEALTHY_BIT *)
  ANDN %M5                (* SC1_FAULT_CONT *)
  ANDN %M4                (* SC1_TRIP *)
  ANDN %M17               (* SC1_AUTO_STOP *)
  AND %M40                (* APP_ON *)
  MPS
  AND( %M13               (* SC1_AUTO_START *)
  OR %I0.7                (* SC1_RUNNING *)
  )
  ST %M23                 (* SC1_ON_AUX *)
  MPP
  ANDF %M23               (* SC1_ON_AUX *)
  S %M4                   (* SC1_TRIP *)
  // as ST:
  //   SC1_ON_AUX := HEALTHY_BIT AND NOT SC1_FAULT_CONT AND NOT SC1_TRIP AND NOT SC1_AUTO_STOP AND APP_ON AND (SC1_AUTO_START OR SC1_RUNNING);
  //   IF HEALTHY_BIT AND NOT SC1_FAULT_CONT AND NOT SC1_TRIP AND NOT SC1_AUTO_STOP AND APP_ON AND FALLING(SC1_ON_AUX) THEN SC1_TRIP := TRUE; END_IF;

// Rung 39: SC1 CONTROL TRIP
  LD %I0.12               (* SC1B_ACTIVE *)
  S %M5                   (* SC1_FAULT_CONT *)
  // as ST:
  //   IF SC1B_ACTIVE THEN SC1_FAULT_CONT := TRUE; END_IF;

// Rung 40: SC1 RUN COIL
  LD %M23                 (* SC1_ON_AUX *)
  ST %Q0.4                (* SC1_ON *)
  // as ST:
  //   SC1_ON := SC1_ON_AUX;

// Rung 41: SC1 CONTROL ON_OFF
  LD %M15                 (* SYY_AUTO_ON *)
  ST %Q0.13               (* SC1_CONT_ON *)
  // as ST:
  //   SC1_CONT_ON := SYY_AUTO_ON;

POU CONVEYOR No3
  (* SectionNumber=9 *)

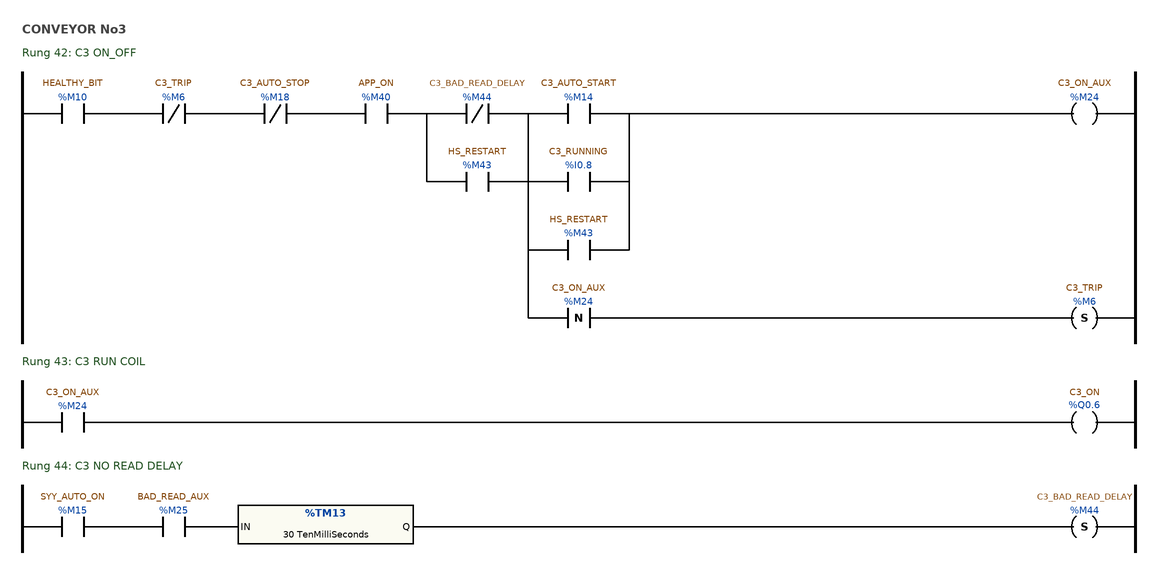

// Rung 42: C3 ON_OFF
  LD %M10                 (* HEALTHY_BIT *)
  ANDN %M6                (* C3_TRIP *)
  ANDN %M18               (* C3_AUTO_STOP *)
  AND %M40                (* APP_ON *)
  AND(N %M44              (* C3_BAD_READ_DELAY *)
  OR %M43                 (* HS_RESTART *)
  )
  MPS
  AND( %M14               (* C3_AUTO_START *)
  OR %I0.8                (* C3_RUNNING *)
  OR %M43                 (* HS_RESTART *)
  )
  ST %M24                 (* C3_ON_AUX *)
  MPP
  ANDF %M24               (* C3_ON_AUX *)
  S %M6                   (* C3_TRIP *)
  // as ST:
  //   C3_ON_AUX := HEALTHY_BIT AND NOT C3_TRIP AND NOT C3_AUTO_STOP AND APP_ON AND (NOT C3_BAD_READ_DELAY OR HS_RESTART) AND (C3_AUTO_START OR C3_RUNNING OR HS_RESTART);
  //   IF HEALTHY_BIT AND NOT C3_TRIP AND NOT C3_AUTO_STOP AND APP_ON AND (NOT C3_BAD_READ_DELAY OR HS_RESTART) AND FALLING(C3_ON_AUX) THEN C3_TRIP := TRUE; END_IF;

// Rung 43: C3 RUN COIL
  LD %M24                 (* C3_ON_AUX *)
  ST %Q0.6                (* C3_ON *)
  // as ST:
  //   C3_ON := C3_ON_AUX;

// Rung 44: C3 NO READ DELAY
  BLK %TM13
  LD %M15                 (* SYY_AUTO_ON *)
  AND %M25                (* BAD_READ_AUX *)
  IN
  OUT_BLK
  LD Q
  S %M44                  (* C3_BAD_READ_DELAY *)
  END_BLK
  // as ST:
  //   %TM13(IN := SYY_AUTO_ON AND BAD_READ_AUX);
  //   IF %TM13.Q THEN C3_BAD_READ_DELAY := TRUE; END_IF;

POU PRODUCT DETECTION
  (* SectionNumber=10 *)

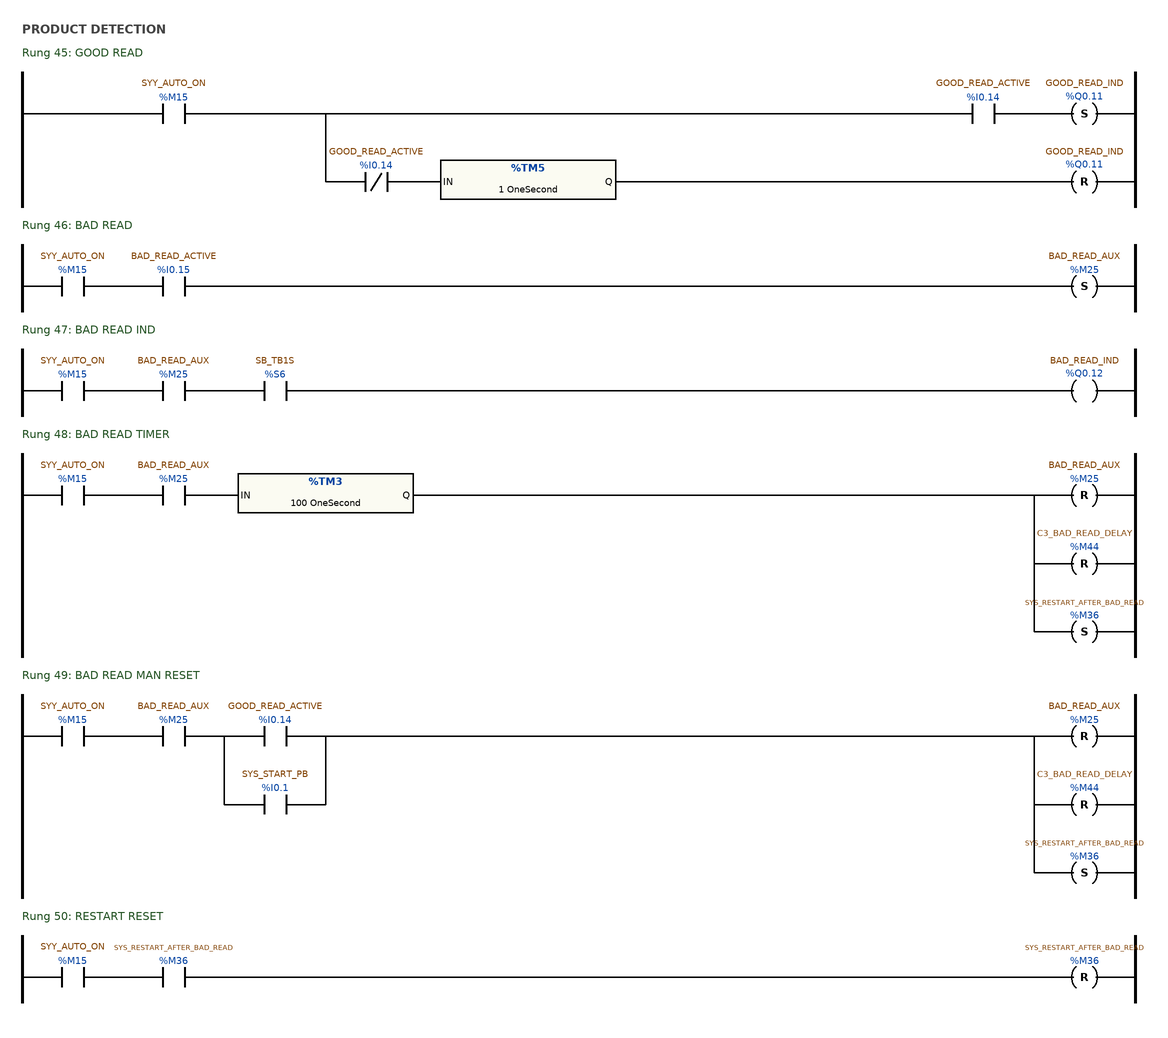

// Rung 45: GOOD READ
  LD 1
  MULTIFB
  LD 1
  AND %M15                (* SYY_AUTO_ON *)
  ST %MW2009:X0
  LD %MW2009:X0
  AND %I0.14              (* GOOD_READ_ACTIVE *)
  S %Q0.11                (* GOOD_READ_IND *)
  BLK %TM5
  LD %MW2009:X0
  ANDN %I0.14             (* GOOD_READ_ACTIVE *)
  IN
  OUT_BLK
  LD Q
  R %Q0.11                (* GOOD_READ_IND *)
  END_BLK
  MULTIFB
  // as ST:
  //   IF SYY_AUTO_ON AND GOOD_READ_ACTIVE THEN GOOD_READ_IND := TRUE; END_IF;
  //   %TM5(IN := SYY_AUTO_ON AND NOT GOOD_READ_ACTIVE);
  //   IF %TM5.Q THEN GOOD_READ_IND := FALSE; END_IF;

// Rung 46: BAD READ
  LD %M15                 (* SYY_AUTO_ON *)
  AND %I0.15              (* BAD_READ_ACTIVE *)
  S %M25                  (* BAD_READ_AUX *)
  // as ST:
  //   IF SYY_AUTO_ON AND BAD_READ_ACTIVE THEN BAD_READ_AUX := TRUE; END_IF;

// Rung 47: BAD READ IND
  LD %M15                 (* SYY_AUTO_ON *)
  AND %M25                (* BAD_READ_AUX *)
  AND %S6                 (* SB_TB1S *)
  ST %Q0.12               (* BAD_READ_IND *)
  // as ST:
  //   BAD_READ_IND := SYY_AUTO_ON AND BAD_READ_AUX AND SB_TB1S;

// Rung 48: BAD READ TIMER
  BLK %TM3
  LD %M15                 (* SYY_AUTO_ON *)
  AND %M25                (* BAD_READ_AUX *)
  IN
  OUT_BLK
  LD Q
  R %M25                  (* BAD_READ_AUX *)
  R %M44                  (* C3_BAD_READ_DELAY *)
  S %M36                  (* SYS_RESTART_AFTER_BAD_READ *)
  END_BLK
  // as ST:
  //   %TM3(IN := SYY_AUTO_ON AND BAD_READ_AUX);
  //   IF %TM3.Q THEN BAD_READ_AUX := FALSE; END_IF;
  //   IF %TM3.Q THEN C3_BAD_READ_DELAY := FALSE; END_IF;
  //   IF %TM3.Q THEN SYS_RESTART_AFTER_BAD_READ := TRUE; END_IF;

// Rung 49: BAD READ MAN RESET
  LD %M15                 (* SYY_AUTO_ON *)
  AND %M25                (* BAD_READ_AUX *)
  AND( %I0.14             (* GOOD_READ_ACTIVE *)
  OR %I0.1                (* SYS_START_PB *)
  )
  R %M25                  (* BAD_READ_AUX *)
  R %M44                  (* C3_BAD_READ_DELAY *)
  S %M36                  (* SYS_RESTART_AFTER_BAD_READ *)
  // as ST:
  //   _t1 := SYY_AUTO_ON AND BAD_READ_AUX AND (GOOD_READ_ACTIVE OR SYS_START_PB);
  //   IF _t1 THEN BAD_READ_AUX := FALSE; END_IF;
  //   IF _t1 THEN C3_BAD_READ_DELAY := FALSE; END_IF;
  //   IF _t1 THEN SYS_RESTART_AFTER_BAD_READ := TRUE; END_IF;

// Rung 50: RESTART RESET
  LD %M15                 (* SYY_AUTO_ON *)
  AND %M36                (* SYS_RESTART_AFTER_BAD_READ *)
  R %M36                  (* SYS_RESTART_AFTER_BAD_READ *)
  // as ST:
  //   IF SYY_AUTO_ON AND SYS_RESTART_AFTER_BAD_READ THEN SYS_RESTART_AFTER_BAD_READ := FALSE; END_IF;

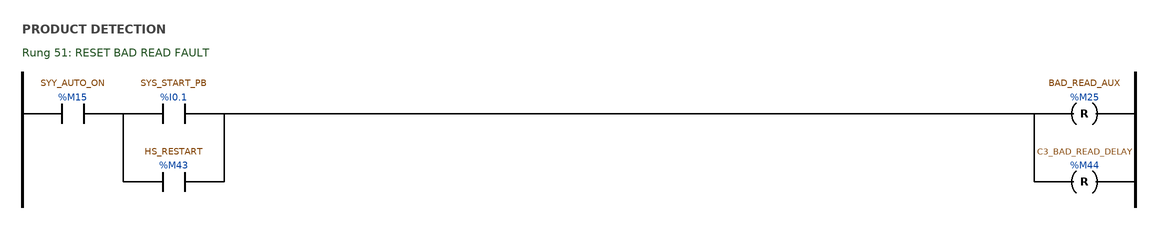

// Rung 51: RESET BAD READ FAULT
  LD %M15                 (* SYY_AUTO_ON *)
  AND( %I0.1              (* SYS_START_PB *)
  OR %M43                 (* HS_RESTART *)
  )
  R %M25                  (* BAD_READ_AUX *)
  R %M44                  (* C3_BAD_READ_DELAY *)
  // as ST:
  //   IF SYY_AUTO_ON AND (SYS_START_PB OR HS_RESTART) THEN BAD_READ_AUX := FALSE; END_IF;
  //   IF SYY_AUTO_ON AND (SYS_START_PB OR HS_RESTART) THEN C3_BAD_READ_DELAY := FALSE; END_IF;

POU C1 PRODUCT SPACING
  (* SectionNumber=11 *)

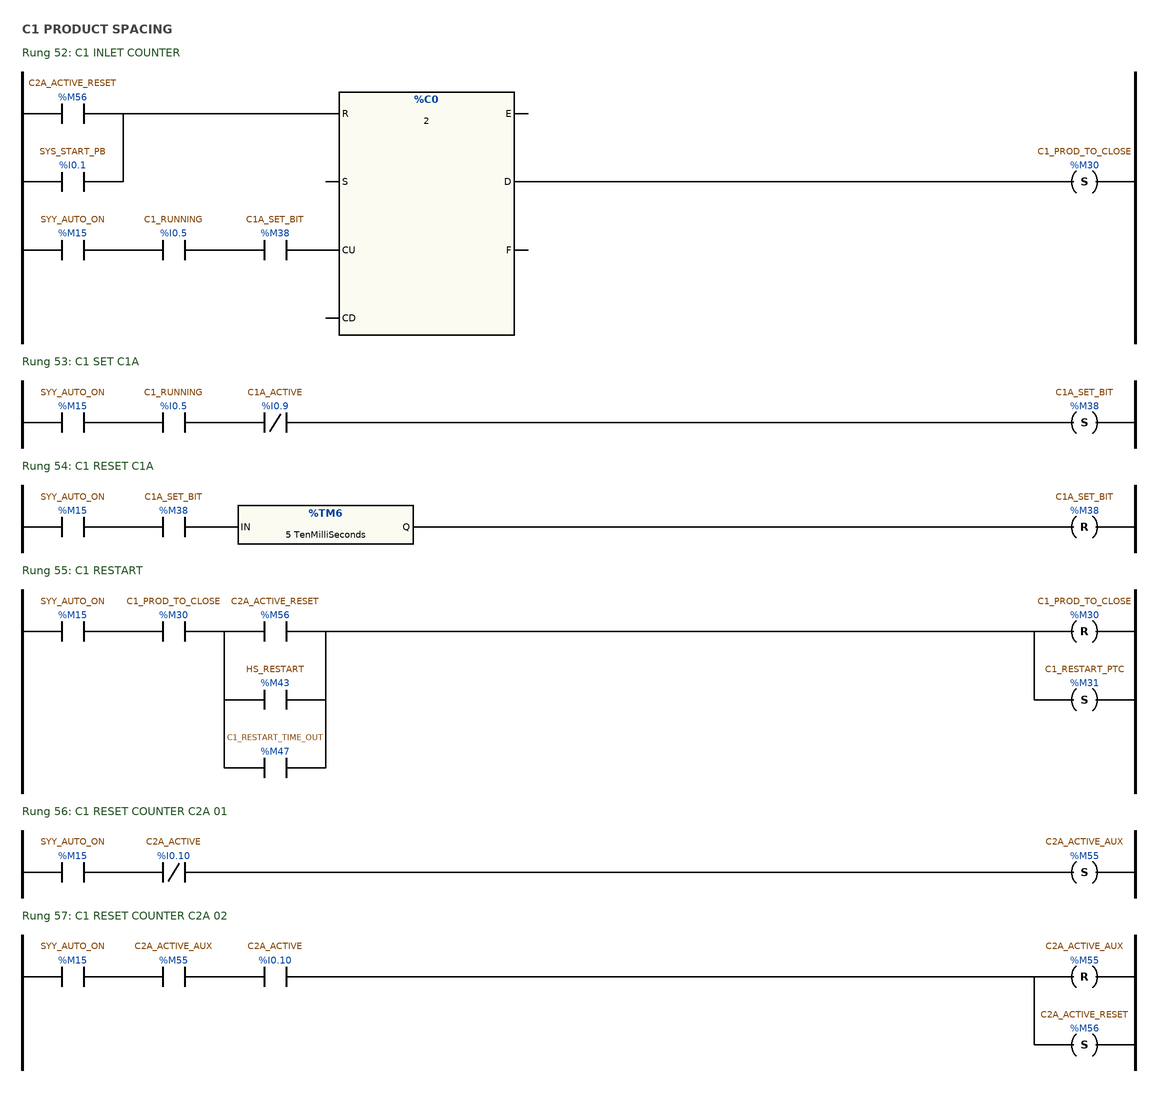

// Rung 52: C1 INLET COUNTER
  BLK %C0
  LD %M56                 (* C2A_ACTIVE_RESET *)
  OR %I0.1                (* SYS_START_PB *)
  R
  LD %M15                 (* SYY_AUTO_ON *)
  AND %I0.5               (* C1_RUNNING *)
  AND %M38                (* C1A_SET_BIT *)
  CU
  OUT_BLK
  LD D
  S %M30                  (* C1_PROD_TO_CLOSE *)
  END_BLK
  // as ST:
  //   %C0(R := C2A_ACTIVE_RESET OR SYS_START_PB, CU := SYY_AUTO_ON AND C1_RUNNING AND C1A_SET_BIT);
  //   IF %C0.D THEN C1_PROD_TO_CLOSE := TRUE; END_IF;

// Rung 53: C1 SET C1A
  LD %M15                 (* SYY_AUTO_ON *)
  AND %I0.5               (* C1_RUNNING *)
  ANDN %I0.9              (* C1A_ACTIVE *)
  S %M38                  (* C1A_SET_BIT *)
  // as ST:
  //   IF SYY_AUTO_ON AND C1_RUNNING AND NOT C1A_ACTIVE THEN C1A_SET_BIT := TRUE; END_IF;

// Rung 54: C1 RESET C1A
  BLK %TM6
  LD %M15                 (* SYY_AUTO_ON *)
  AND %M38                (* C1A_SET_BIT *)
  IN
  OUT_BLK
  LD Q
  R %M38                  (* C1A_SET_BIT *)
  END_BLK
  // as ST:
  //   %TM6(IN := SYY_AUTO_ON AND C1A_SET_BIT);
  //   IF %TM6.Q THEN C1A_SET_BIT := FALSE; END_IF;

// Rung 55: C1 RESTART
  LD %M15                 (* SYY_AUTO_ON *)
  AND %M30                (* C1_PROD_TO_CLOSE *)
  AND( %M56               (* C2A_ACTIVE_RESET *)
  OR %M43                 (* HS_RESTART *)
  OR %M47                 (* C1_RESTART_TIME_OUT *)
  )
  R %M30                  (* C1_PROD_TO_CLOSE *)
  S %M31                  (* C1_RESTART_PTC *)
  // as ST:
  //   _t1 := SYY_AUTO_ON AND C1_PROD_TO_CLOSE AND (C2A_ACTIVE_RESET OR HS_RESTART OR C1_RESTART_TIME_OUT);
  //   IF _t1 THEN C1_PROD_TO_CLOSE := FALSE; END_IF;
  //   IF _t1 THEN C1_RESTART_PTC := TRUE; END_IF;

// Rung 56: C1 RESET COUNTER C2A 01
  LD %M15                 (* SYY_AUTO_ON *)
  ANDN %I0.10             (* C2A_ACTIVE *)
  S %M55                  (* C2A_ACTIVE_AUX *)
  // as ST:
  //   IF SYY_AUTO_ON AND NOT C2A_ACTIVE THEN C2A_ACTIVE_AUX := TRUE; END_IF;

// Rung 57: C1 RESET COUNTER C2A 02
  LD %M15                 (* SYY_AUTO_ON *)
  AND %M55                (* C2A_ACTIVE_AUX *)
  AND %I0.10              (* C2A_ACTIVE *)
  R %M55                  (* C2A_ACTIVE_AUX *)
  S %M56                  (* C2A_ACTIVE_RESET *)
  // as ST:
  //   _t1 := SYY_AUTO_ON AND C2A_ACTIVE_AUX AND C2A_ACTIVE;
  //   IF _t1 THEN C2A_ACTIVE_AUX := FALSE; END_IF;
  //   IF _t1 THEN C2A_ACTIVE_RESET := TRUE; END_IF;

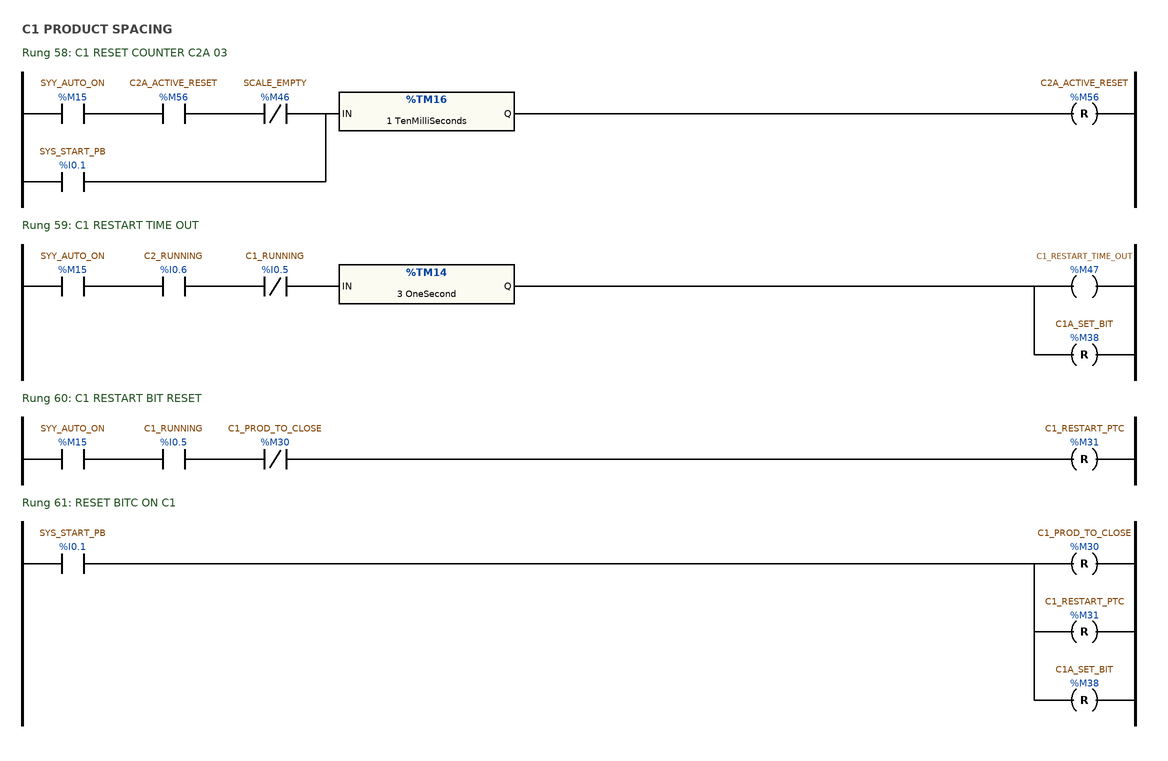

// Rung 58: C1 RESET COUNTER C2A 03
  BLK %TM16
  LD %M15                 (* SYY_AUTO_ON *)
  AND %M56                (* C2A_ACTIVE_RESET *)
  ANDN %M46               (* SCALE_EMPTY *)
  OR %I0.1                (* SYS_START_PB *)
  IN
  OUT_BLK
  LD Q
  R %M56                  (* C2A_ACTIVE_RESET *)
  END_BLK
  // as ST:
  //   %TM16(IN := SYY_AUTO_ON AND C2A_ACTIVE_RESET AND NOT SCALE_EMPTY OR SYS_START_PB);
  //   IF %TM16.Q THEN C2A_ACTIVE_RESET := FALSE; END_IF;

// Rung 59: C1 RESTART TIME OUT
  BLK %TM14
  LD %M15                 (* SYY_AUTO_ON *)
  AND %I0.6               (* C2_RUNNING *)
  ANDN %I0.5              (* C1_RUNNING *)
  IN
  OUT_BLK
  LD Q
  ST %M47                 (* C1_RESTART_TIME_OUT *)
  R %M38                  (* C1A_SET_BIT *)
  END_BLK
  // as ST:
  //   %TM14(IN := SYY_AUTO_ON AND C2_RUNNING AND NOT C1_RUNNING);
  //   C1_RESTART_TIME_OUT := %TM14.Q;
  //   IF %TM14.Q THEN C1A_SET_BIT := FALSE; END_IF;

// Rung 60: C1 RESTART BIT RESET
  LD %M15                 (* SYY_AUTO_ON *)
  AND %I0.5               (* C1_RUNNING *)
  ANDN %M30               (* C1_PROD_TO_CLOSE *)
  R %M31                  (* C1_RESTART_PTC *)
  // as ST:
  //   IF SYY_AUTO_ON AND C1_RUNNING AND NOT C1_PROD_TO_CLOSE THEN C1_RESTART_PTC := FALSE; END_IF;

// Rung 61: RESET BITC ON C1
  LD %I0.1                (* SYS_START_PB *)
  R %M30                  (* C1_PROD_TO_CLOSE *)
  R %M31                  (* C1_RESTART_PTC *)
  R %M38                  (* C1A_SET_BIT *)
  // as ST:
  //   IF SYS_START_PB THEN C1_PROD_TO_CLOSE := FALSE; END_IF;
  //   IF SYS_START_PB THEN C1_RESTART_PTC := FALSE; END_IF;
  //   IF SYS_START_PB THEN C1A_SET_BIT := FALSE; END_IF;

POU C2 PRODUCT TO CLOSED
  (* SectionNumber=12 *)

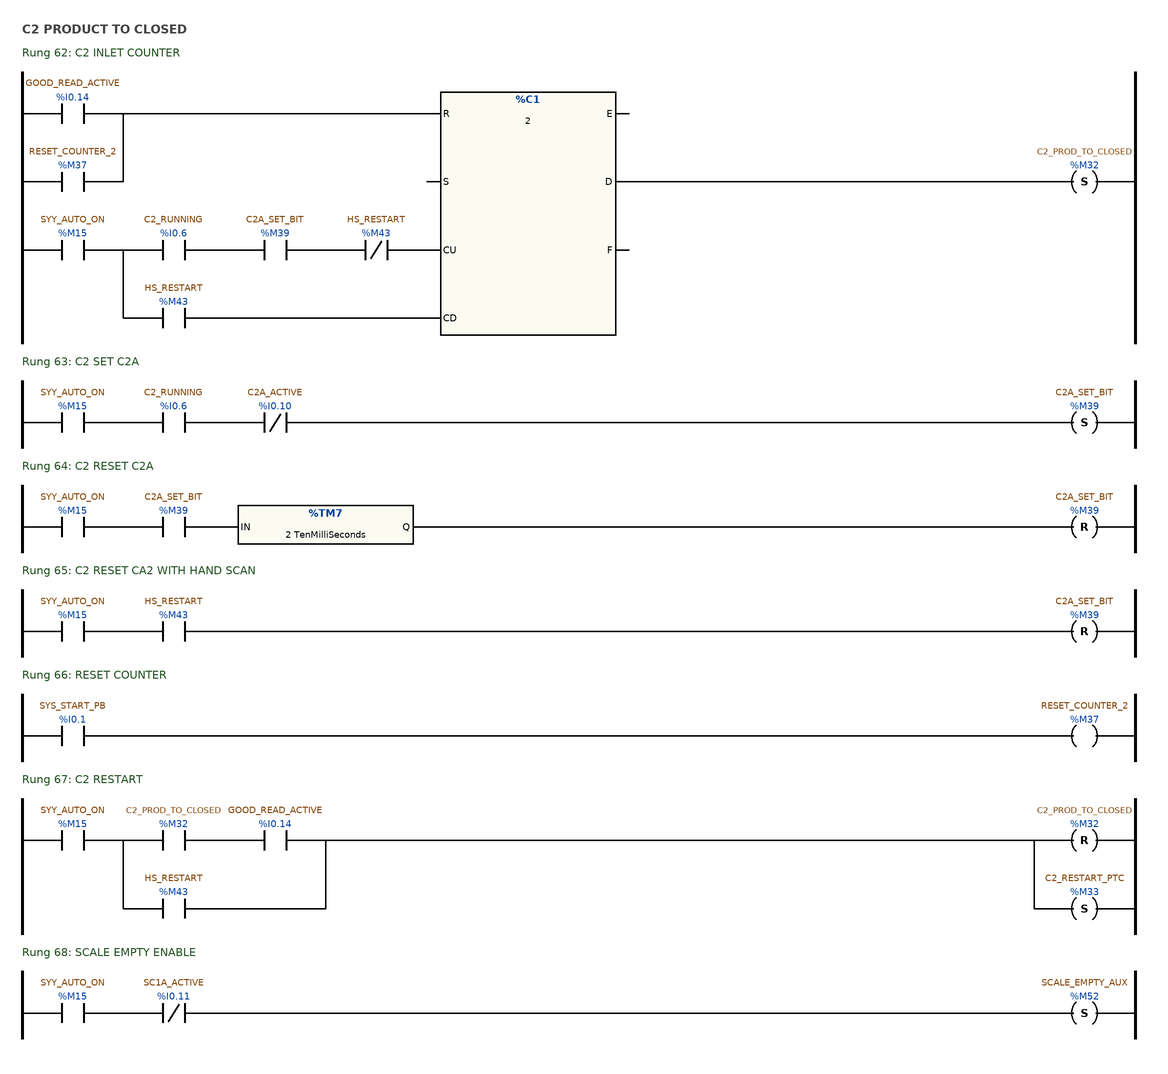

// Rung 62: C2 INLET COUNTER
  BLK %C1
  LD %I0.14               (* GOOD_READ_ACTIVE *)
  OR %M37                 (* RESET_COUNTER_2 *)
  R
  LD %M15                 (* SYY_AUTO_ON *)
  MPS
  AND %I0.6               (* C2_RUNNING *)
  AND %M39                (* C2A_SET_BIT *)
  ANDN %M43               (* HS_RESTART *)
  CU
  MPP
  AND %M43                (* HS_RESTART *)
  CD
  OUT_BLK
  LD D
  S %M32                  (* C2_PROD_TO_CLOSED *)
  END_BLK
  // as ST:
  //   %C1(R := GOOD_READ_ACTIVE OR RESET_COUNTER_2, CU := SYY_AUTO_ON AND C2_RUNNING AND C2A_SET_BIT AND NOT HS_RESTART, CD := SYY_AUTO_ON AND HS_RESTART);
  //   IF %C1.D THEN C2_PROD_TO_CLOSED := TRUE; END_IF;

// Rung 63: C2 SET C2A
  LD %M15                 (* SYY_AUTO_ON *)
  AND %I0.6               (* C2_RUNNING *)
  ANDN %I0.10             (* C2A_ACTIVE *)
  S %M39                  (* C2A_SET_BIT *)
  // as ST:
  //   IF SYY_AUTO_ON AND C2_RUNNING AND NOT C2A_ACTIVE THEN C2A_SET_BIT := TRUE; END_IF;

// Rung 64: C2 RESET C2A
  BLK %TM7
  LD %M15                 (* SYY_AUTO_ON *)
  AND %M39                (* C2A_SET_BIT *)
  IN
  OUT_BLK
  LD Q
  R %M39                  (* C2A_SET_BIT *)
  END_BLK
  // as ST:
  //   %TM7(IN := SYY_AUTO_ON AND C2A_SET_BIT);
  //   IF %TM7.Q THEN C2A_SET_BIT := FALSE; END_IF;

// Rung 65: C2 RESET CA2 WITH HAND SCAN
  LD %M15                 (* SYY_AUTO_ON *)
  AND %M43                (* HS_RESTART *)
  R %M39                  (* C2A_SET_BIT *)
  // as ST:
  //   IF SYY_AUTO_ON AND HS_RESTART THEN C2A_SET_BIT := FALSE; END_IF;

// Rung 66: RESET COUNTER
  LD %I0.1                (* SYS_START_PB *)
  ST %M37                 (* RESET_COUNTER_2 *)
  // as ST:
  //   RESET_COUNTER_2 := SYS_START_PB;

// Rung 67: C2 RESTART
  LD %M15                 (* SYY_AUTO_ON *)
  AND( %M32               (* C2_PROD_TO_CLOSED *)
  AND %I0.14              (* GOOD_READ_ACTIVE *)
  OR %M43                 (* HS_RESTART *)
  )
  R %M32                  (* C2_PROD_TO_CLOSED *)
  S %M33                  (* C2_RESTART_PTC *)
  // as ST:
  //   _t1 := SYY_AUTO_ON AND (C2_PROD_TO_CLOSED AND GOOD_READ_ACTIVE OR HS_RESTART);
  //   IF _t1 THEN C2_PROD_TO_CLOSED := FALSE; END_IF;
  //   IF _t1 THEN C2_RESTART_PTC := TRUE; END_IF;

// Rung 68: SCALE EMPTY ENABLE
  LD %M15                 (* SYY_AUTO_ON *)
  ANDN %I0.11             (* SC1A_ACTIVE *)
  S %M52                  (* SCALE_EMPTY_AUX *)
  // as ST:
  //   IF SYY_AUTO_ON AND NOT SC1A_ACTIVE THEN SCALE_EMPTY_AUX := TRUE; END_IF;

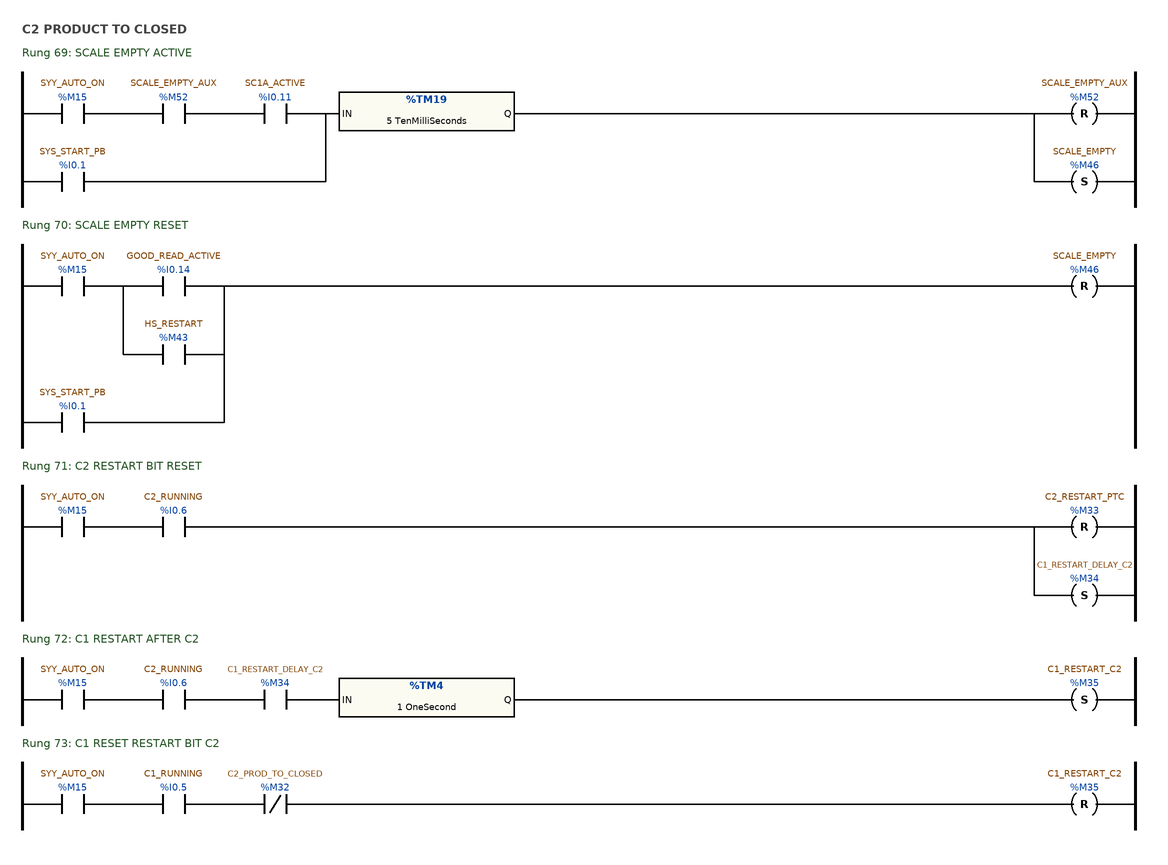

// Rung 69: SCALE EMPTY ACTIVE
  BLK %TM19
  LD %M15                 (* SYY_AUTO_ON *)
  AND %M52                (* SCALE_EMPTY_AUX *)
  AND %I0.11              (* SC1A_ACTIVE *)
  OR %I0.1                (* SYS_START_PB *)
  IN
  OUT_BLK
  LD Q
  R %M52                  (* SCALE_EMPTY_AUX *)
  S %M46                  (* SCALE_EMPTY *)
  END_BLK
  // as ST:
  //   %TM19(IN := SYY_AUTO_ON AND SCALE_EMPTY_AUX AND SC1A_ACTIVE OR SYS_START_PB);
  //   IF %TM19.Q THEN SCALE_EMPTY_AUX := FALSE; END_IF;
  //   IF %TM19.Q THEN SCALE_EMPTY := TRUE; END_IF;

// Rung 70: SCALE EMPTY RESET
  LD %M15                 (* SYY_AUTO_ON *)
  AND( %I0.14             (* GOOD_READ_ACTIVE *)
  OR %M43                 (* HS_RESTART *)
  )
  OR %I0.1                (* SYS_START_PB *)
  R %M46                  (* SCALE_EMPTY *)
  // as ST:
  //   IF SYY_AUTO_ON AND (GOOD_READ_ACTIVE OR HS_RESTART) OR SYS_START_PB THEN SCALE_EMPTY := FALSE; END_IF;

// Rung 71: C2 RESTART BIT RESET
  LD %M15                 (* SYY_AUTO_ON *)
  AND %I0.6               (* C2_RUNNING *)
  R %M33                  (* C2_RESTART_PTC *)
  S %M34                  (* C1_RESTART_DELAY_C2 *)
  // as ST:
  //   IF SYY_AUTO_ON AND C2_RUNNING THEN C2_RESTART_PTC := FALSE; END_IF;
  //   IF SYY_AUTO_ON AND C2_RUNNING THEN C1_RESTART_DELAY_C2 := TRUE; END_IF;

// Rung 72: C1 RESTART AFTER C2
  BLK %TM4
  LD %M15                 (* SYY_AUTO_ON *)
  AND %I0.6               (* C2_RUNNING *)
  AND %M34                (* C1_RESTART_DELAY_C2 *)
  IN
  OUT_BLK
  LD Q
  S %M35                  (* C1_RESTART_C2 *)
  END_BLK
  // as ST:
  //   %TM4(IN := SYY_AUTO_ON AND C2_RUNNING AND C1_RESTART_DELAY_C2);
  //   IF %TM4.Q THEN C1_RESTART_C2 := TRUE; END_IF;

// Rung 73: C1 RESET RESTART BIT C2
  LD %M15                 (* SYY_AUTO_ON *)
  AND %I0.5               (* C1_RUNNING *)
  ANDN %M32               (* C2_PROD_TO_CLOSED *)
  R %M35                  (* C1_RESTART_C2 *)
  // as ST:
  //   IF SYY_AUTO_ON AND C1_RUNNING AND NOT C2_PROD_TO_CLOSED THEN C1_RESTART_C2 := FALSE; END_IF;

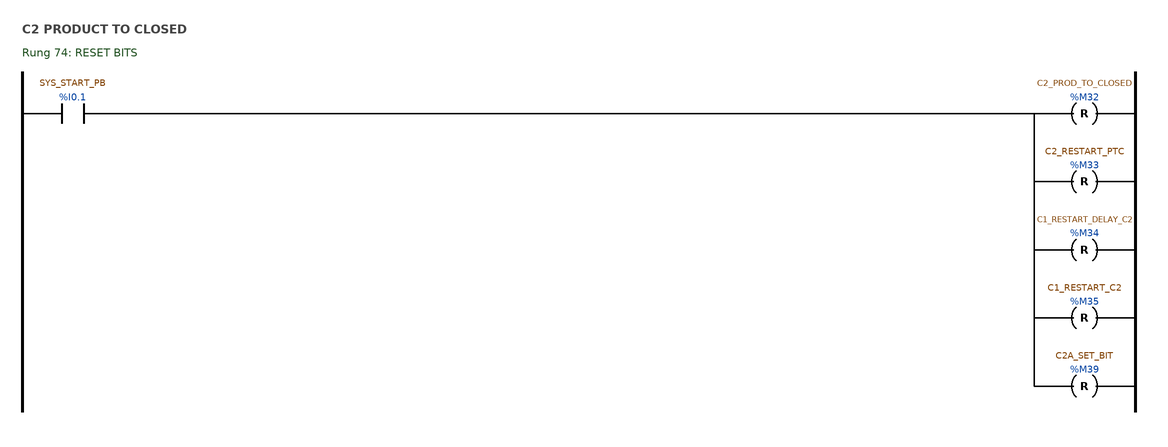

// Rung 74: RESET BITS
  LD %I0.1                (* SYS_START_PB *)
  R %M32                  (* C2_PROD_TO_CLOSED *)
  R %M33                  (* C2_RESTART_PTC *)
  R %M34                  (* C1_RESTART_DELAY_C2 *)
  R %M35                  (* C1_RESTART_C2 *)
  R %M39                  (* C2A_SET_BIT *)
  // as ST:
  //   IF SYS_START_PB THEN C2_PROD_TO_CLOSED := FALSE; END_IF;
  //   IF SYS_START_PB THEN C2_RESTART_PTC := FALSE; END_IF;
  //   IF SYS_START_PB THEN C1_RESTART_DELAY_C2 := FALSE; END_IF;
  //   IF SYS_START_PB THEN C1_RESTART_C2 := FALSE; END_IF;
  //   IF SYS_START_PB THEN C2A_SET_BIT := FALSE; END_IF;

POU COMUNICATION OUT
  (* SectionNumber=13 *)

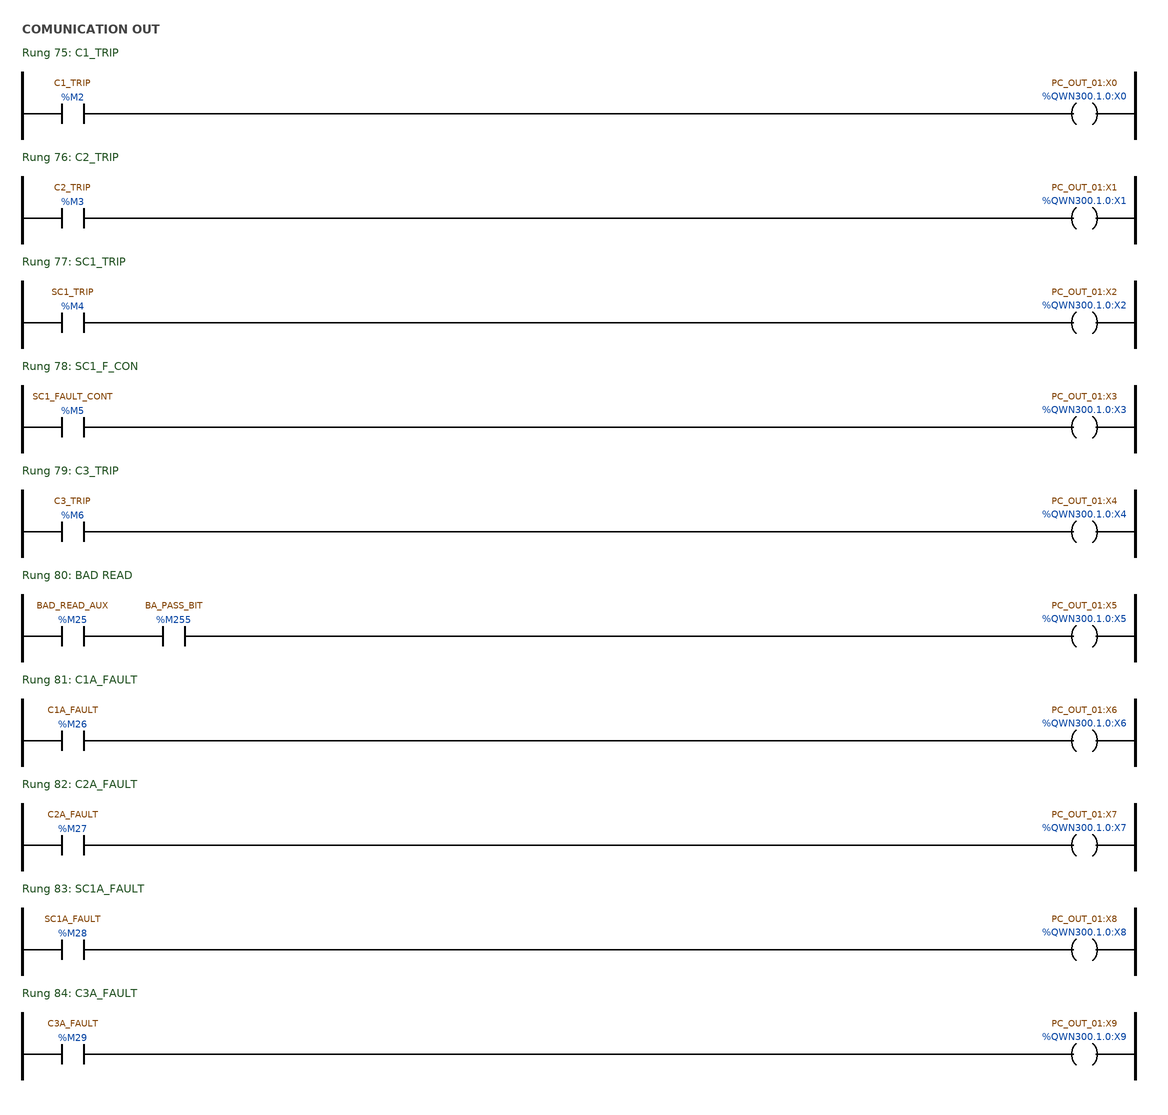

// Rung 75: C1_TRIP
  LD %M2                  (* C1_TRIP *)
  ST %QWN300.1.0:X0       (* PC_OUT_01 *)
  // as ST:
  //   PC_OUT_01:X0 := C1_TRIP;

// Rung 76: C2_TRIP
  LD %M3                  (* C2_TRIP *)
  ST %QWN300.1.0:X1       (* PC_OUT_01 *)
  // as ST:
  //   PC_OUT_01:X1 := C2_TRIP;

// Rung 77: SC1_TRIP
  LD %M4                  (* SC1_TRIP *)
  ST %QWN300.1.0:X2       (* PC_OUT_01 *)
  // as ST:
  //   PC_OUT_01:X2 := SC1_TRIP;

// Rung 78: SC1_F_CON
  LD %M5                  (* SC1_FAULT_CONT *)
  ST %QWN300.1.0:X3       (* PC_OUT_01 *)
  // as ST:
  //   PC_OUT_01:X3 := SC1_FAULT_CONT;

// Rung 79: C3_TRIP
  LD %M6                  (* C3_TRIP *)
  ST %QWN300.1.0:X4       (* PC_OUT_01 *)
  // as ST:
  //   PC_OUT_01:X4 := C3_TRIP;

// Rung 80: BAD READ
  LD %M25                 (* BAD_READ_AUX *)
  AND %M255               (* BA_PASS_BIT *)
  ST %QWN300.1.0:X5       (* PC_OUT_01 *)
  // as ST:
  //   PC_OUT_01:X5 := BAD_READ_AUX AND BA_PASS_BIT;

// Rung 81: C1A_FAULT
  LD %M26                 (* C1A_FAULT *)
  ST %QWN300.1.0:X6       (* PC_OUT_01 *)
  // as ST:
  //   PC_OUT_01:X6 := C1A_FAULT;

// Rung 82: C2A_FAULT
  LD %M27                 (* C2A_FAULT *)
  ST %QWN300.1.0:X7       (* PC_OUT_01 *)
  // as ST:
  //   PC_OUT_01:X7 := C2A_FAULT;

// Rung 83: SC1A_FAULT
  LD %M28                 (* SC1A_FAULT *)
  ST %QWN300.1.0:X8       (* PC_OUT_01 *)
  // as ST:
  //   PC_OUT_01:X8 := SC1A_FAULT;

// Rung 84: C3A_FAULT
  LD %M29                 (* C3A_FAULT *)
  ST %QWN300.1.0:X9       (* PC_OUT_01 *)
  // as ST:
  //   PC_OUT_01:X9 := C3A_FAULT;

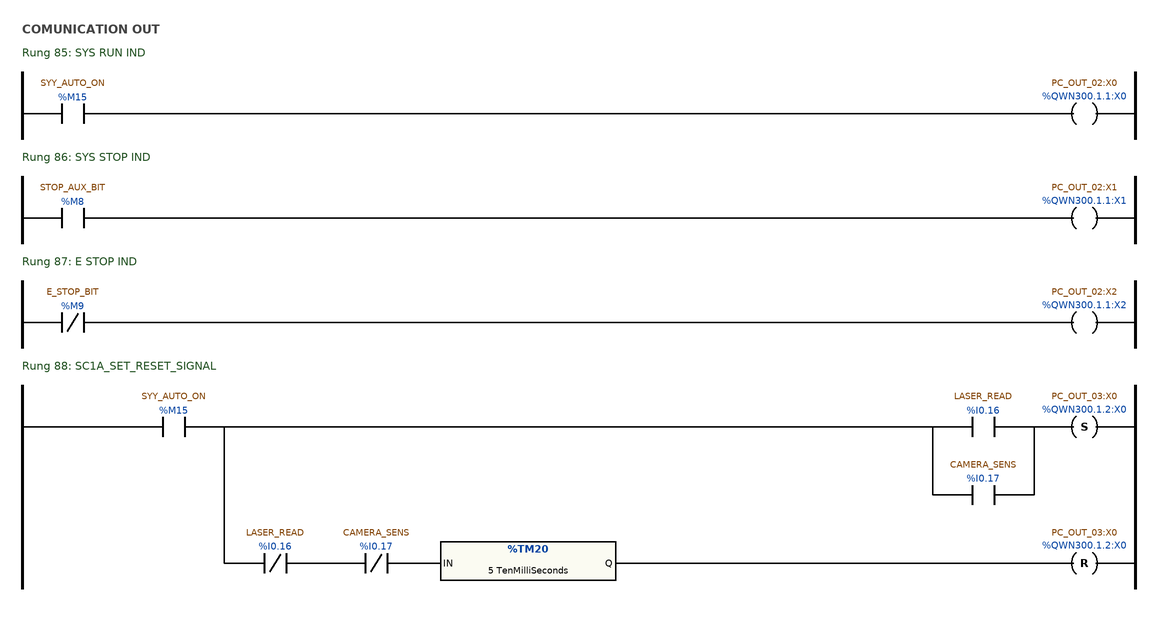

// Rung 85: SYS RUN IND
  LD %M15                 (* SYY_AUTO_ON *)
  ST %QWN300.1.1:X0       (* PC_OUT_02 *)
  // as ST:
  //   PC_OUT_02:X0 := SYY_AUTO_ON;

// Rung 86: SYS STOP IND
  LD %M8                  (* STOP_AUX_BIT *)
  ST %QWN300.1.1:X1       (* PC_OUT_02 *)
  // as ST:
  //   PC_OUT_02:X1 := STOP_AUX_BIT;

// Rung 87: E STOP IND
  LDN %M9                 (* E_STOP_BIT *)
  ST %QWN300.1.1:X2       (* PC_OUT_02 *)
  // as ST:
  //   PC_OUT_02:X2 := NOT E_STOP_BIT;

// Rung 88: SC1A_SET_RESET_SIGNAL
  LD 1
  MULTIFB
  LD 1
  AND %M15                (* SYY_AUTO_ON *)
  ST %MW2009:X0
  LD %MW2009:X0
  AND( %I0.16             (* LASER_READ *)
  OR %I0.17               (* CAMERA_SENS *)
  )
  S %QWN300.1.2:X0        (* PC_OUT_03 *)
  BLK %TM20
  LD %MW2009:X0
  ANDN %I0.16             (* LASER_READ *)
  ANDN %I0.17             (* CAMERA_SENS *)
  IN
  OUT_BLK
  LD Q
  R %QWN300.1.2:X0        (* PC_OUT_03 *)
  END_BLK
  MULTIFB
  // as ST:
  //   IF SYY_AUTO_ON AND (LASER_READ OR CAMERA_SENS) THEN PC_OUT_03:X0 := TRUE; END_IF;
  //   %TM20(IN := SYY_AUTO_ON AND NOT LASER_READ AND NOT CAMERA_SENS);
  //   IF %TM20.Q THEN PC_OUT_03:X0 := FALSE; END_IF;

POU COMUNICATION IN
  (* SectionNumber=14 *)

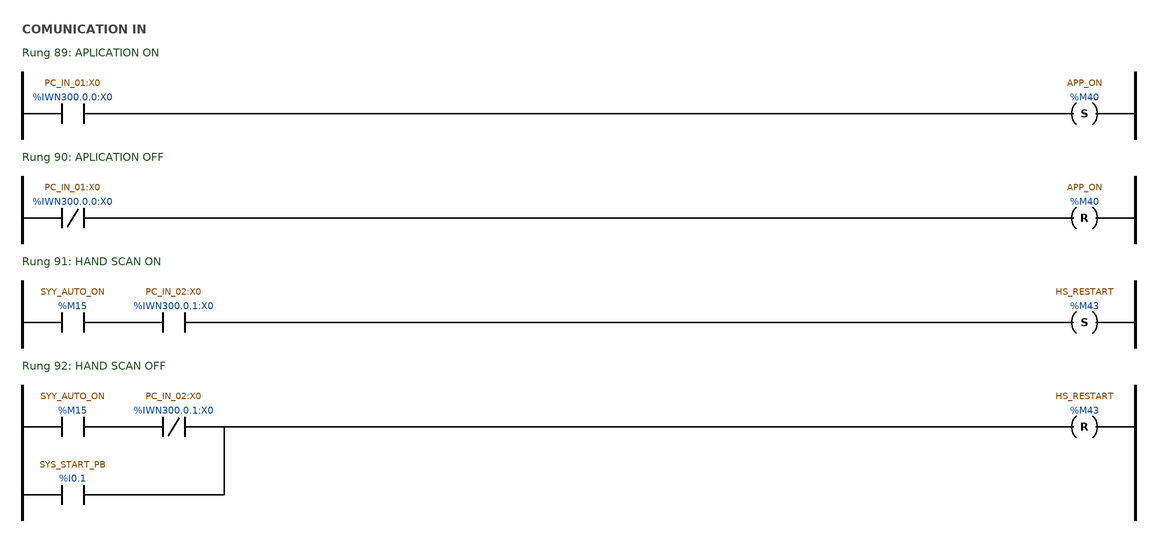

// Rung 89: APLICATION ON
  LD %IWN300.0.0:X0       (* PC_IN_01 *)
  S %M40                  (* APP_ON *)
  // as ST:
  //   IF PC_IN_01:X0 THEN APP_ON := TRUE; END_IF;

// Rung 90: APLICATION OFF
  LDN %IWN300.0.0:X0      (* PC_IN_01 *)
  R %M40                  (* APP_ON *)
  // as ST:
  //   IF NOT PC_IN_01:X0 THEN APP_ON := FALSE; END_IF;

// Rung 91: HAND SCAN ON
  LD %M15                 (* SYY_AUTO_ON *)
  AND %IWN300.0.1:X0      (* PC_IN_02 *)
  S %M43                  (* HS_RESTART *)
  // as ST:
  //   IF SYY_AUTO_ON AND PC_IN_02:X0 THEN HS_RESTART := TRUE; END_IF;

// Rung 92: HAND SCAN OFF
  LD %M15                 (* SYY_AUTO_ON *)
  ANDN %IWN300.0.1:X0     (* PC_IN_02 *)
  OR %I0.1                (* SYS_START_PB *)
  R %M43                  (* HS_RESTART *)
  // as ST:
  //   IF SYY_AUTO_ON AND NOT PC_IN_02:X0 OR SYS_START_PB THEN HS_RESTART := FALSE; END_IF;

POU COM PORT 
  (* SectionNumber=15 *)

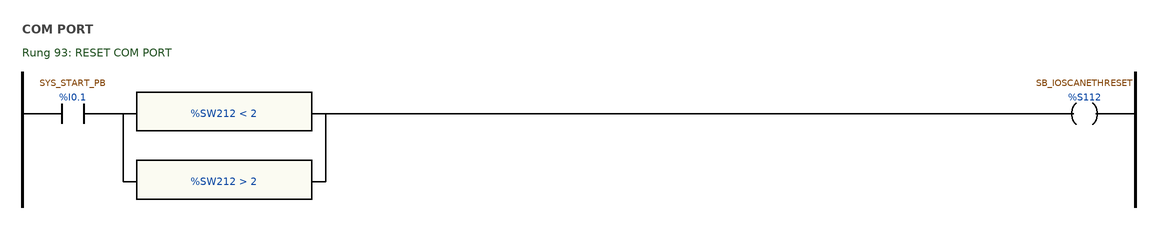

// Rung 93: RESET COM PORT
  LD %I0.1                (* SYS_START_PB *)
  AND( [ %SW212 < 2 ]     (* SW_IOSCANETHSTATUS *)
  OR [ %SW212 > 2 ]       (* SW_IOSCANETHSTATUS *)
  )
  ST %S112                (* SB_IOSCANETHRESET *)
  // as ST:
  //   SB_IOSCANETHRESET := SYS_START_PB AND (SW_IOSCANETHSTATUS < 2 OR SW_IOSCANETHSTATUS > 2);

POU COOLING FAN & INTERFACE
  (* SectionNumber=16 *)

